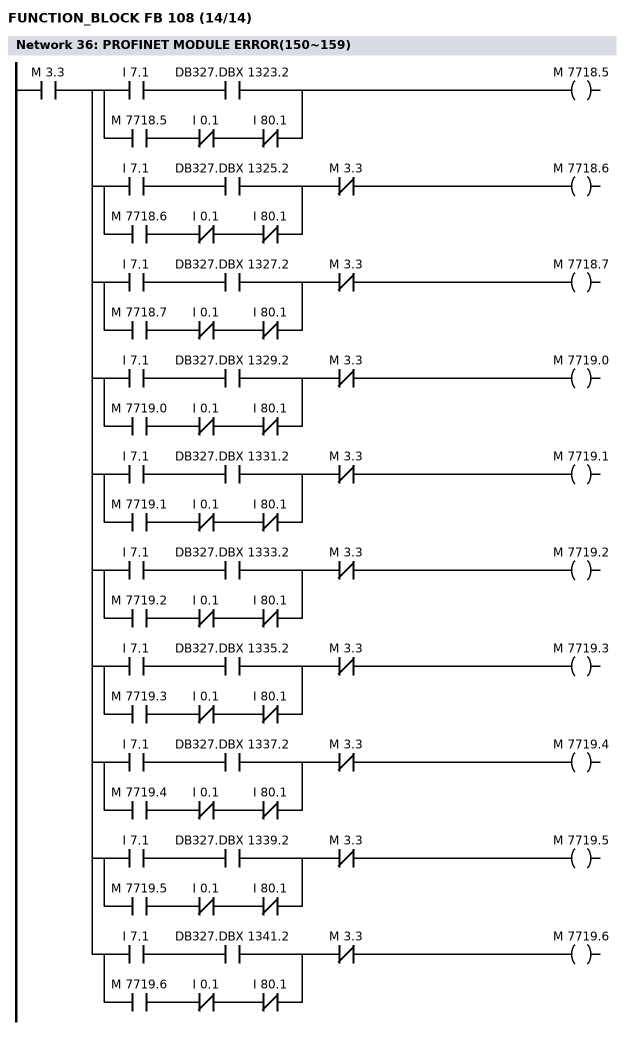

      A     M      3.3;
      =     L      0.0;
      A     L      0.0;
      A(    ;
      A     I      7.1;
      A     DB327.DBX 1323.2;
      O     ;
      A     M   7718.5;
      AN    I      0.1;
      AN    I     80.1;
      )     ;
      =     M   7718.5;
      A     L      0.0;
      A(    ;
      A     I      7.1;
      A     DB327.DBX 1325.2;
      O     ;
      A     M   7718.6;
      AN    I      0.1;
      AN    I     80.1;
      )     ;
      AN    M      3.3;
      =     M   7718.6;
      A     L      0.0;
      A(    ;
      A     I      7.1;
      A     DB327.DBX 1327.2;
      O     ;
      A     M   7718.7;
      AN    I      0.1;
      AN    I     80.1;
      )     ;
      AN    M      3.3;
      =     M   7718.7;
      A     L      0.0;
      A(    ;
      A     I      7.1;
      A     DB327.DBX 1329.2;
      O     ;
      A     M   7719.0;
      AN    I      0.1;
      AN    I     80.1;
      )     ;
      AN    M      3.3;
      =     M   7719.0;
      A     L      0.0;
      A(    ;
      A     I      7.1;
      A     DB327.DBX 1331.2;
      O     ;
      A     M   7719.1;
      AN    I      0.1;
      AN    I     80.1;
      )     ;
      AN    M      3.3;
      =     M   7719.1;
      A     L      0.0;
      A(    ;
      A     I      7.1;
      A     DB327.DBX 1333.2;
      O     ;
      A     M   7719.2;
      AN    I      0.1;
      AN    I     80.1;
      )     ;
      AN    M      3.3;
      =     M   7719.2;
      A     L      0.0;
      A(    ;
      A     I      7.1;
      A     DB327.DBX 1335.2;
      O     ;
      A     M   7719.3;
      AN    I      0.1;
      AN    I     80.1;
      )     ;
      AN    M      3.3;
      =     M   7719.3;
      A     L      0.0;
      A(    ;
      A     I      7.1;
      A     DB327.DBX 1337.2;
      O     ;
      A     M   7719.4;
      AN    I      0.1;
      AN    I     80.1;
      )     ;
      AN    M      3.3;
      =     M   7719.4;
      A     L      0.0;
      A(    ;
      A     I      7.1;
      A     DB327.DBX 1339.2;
      O     ;
      A     M   7719.5;
      AN    I      0.1;
      AN    I     80.1;
      )     ;
      AN    M      3.3;
      =     M   7719.5;
      A     L      0.0;
      A(    ;
      A     I      7.1;
      A     DB327.DBX 1341.2;
      O     ;
      A     M   7719.6;
      AN    I      0.1;
      AN    I     80.1;
      )     ;
      AN    M      3.3;
      =     M   7719.6;
END_FUNCTION_BLOCK

DATA_BLOCK DB 108
TITLE =
VERSION : 0.0

 FB 108
BEGIN
END_DATA_BLOCK

FUNCTION_BLOCK FB 110
TITLE =
VERSION : 0.1


VAR
  S705_MODE : FB 402;
END_VAR
BEGIN
NETWORK
TITLE =
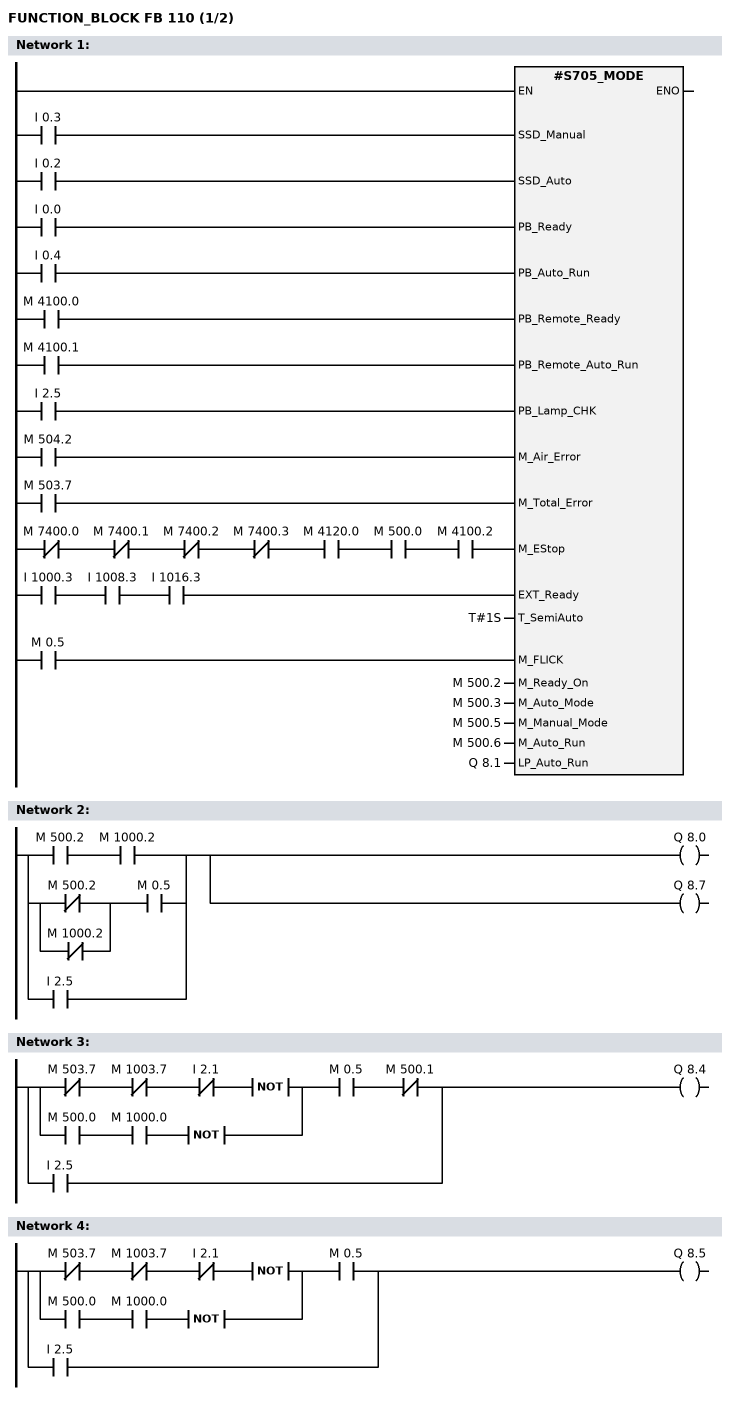

      A     I      0.3;
      =     L      0.0;
      BLD   103;
      A     I      0.2;
      =     L      0.1;
      BLD   103;
      A     I      0.0;
      =     L      0.2;
      BLD   103;
      A     I      0.4;
      =     L      0.3;
      BLD   103;
      A     M   4100.0;
      =     L      0.4;
      BLD   103;
      A     M   4100.1;
      =     L      0.5;
      BLD   103;
      A     I      2.5;
      =     L      0.6;
      BLD   103;
      A     M    504.2;
      =     L      0.7;
      BLD   103;
      A     M    503.7;
      =     L      1.1;
      BLD   103;
      AN    M   7400.0;
      AN    M   7400.1;
      AN    M   7400.2;
      AN    M   7400.3;
      A     M   4120.0;
      A     M    500.0;
      A     M   4100.2;
      =     L      1.2;
      BLD   103;
      A     I   1000.3;
      A     I   1008.3;
      A     I   1016.3;
      =     L      1.3;
      BLD   103;
      A     M      0.5;
      =     L      1.5;
      BLD   103;
      CALL #S705_MODE (
           SSD_Manual               := L      0.0,
           SSD_Auto                 := L      0.1,
           PB_Ready                 := L      0.2,
           PB_Auto_Run              := L      0.3,
           PB_Remote_Ready          := L      0.4,
           PB_Remote_Auto_Run       := L      0.5,
           PB_Lamp_CHK              := L      0.6,
           M_Air_Error              := L      0.7,
           M_Total_Error            := L      1.1,
           M_EStop                  := L      1.2,
           EXT_Ready                := L      1.3,
           T_SemiAuto               := T#1S,
           M_FLICK                  := L      1.5,
           M_Ready_On               := M    500.2,
           M_Auto_Mode              := M    500.3,
           M_Manual_Mode            := M    500.5,
           M_Auto_Run               := M    500.6,
           LP_Auto_Run              := Q      8.1);
      NOP   0;
NETWORK
TITLE =

      A     M    500.2;
      A     M   1000.2;
      O     ;
      A(    ;
      ON    M    500.2;
      ON    M   1000.2;
      )     ;
      A     M      0.5;
      O     I      2.5;
      =     Q      8.0;
      =     Q      8.7;
NETWORK
TITLE =

      A(    ;
      AN    M    503.7;
      AN    M   1003.7;
      AN    I      2.1;
      NOT   ;
      O(    ;
      A     M    500.0;
      A     M   1000.0;
      NOT   ;
      )     ;
      )     ;
      A     M      0.5;
      AN    M    500.1;
      O     I      2.5;
      =     Q      8.4;
NETWORK
TITLE =

      A(    ;
      AN    M    503.7;
      AN    M   1003.7;
      AN    I      2.1;
      NOT   ;
      O(    ;
      A     M    500.0;
      A     M   1000.0;
      NOT   ;
      )     ;
      )     ;
      A     M      0.5;
      O     I      2.5;
      =     Q      8.5;
NETWORK
TITLE =
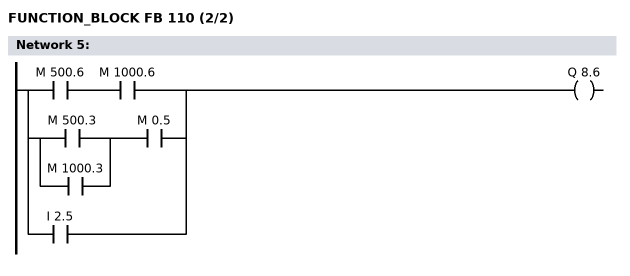

      A     M    500.6;
      A     M   1000.6;
      O     ;
      A(    ;
      O     M    500.3;
      O     M   1000.3;
      )     ;
      A     M      0.5;
      O     I      2.5;
      =     Q      8.6;
END_FUNCTION_BLOCK

DATA_BLOCK DB 110
TITLE =
VERSION : 0.0

 FB 110
BEGIN
   S705_MODE.SSD_Manual := FALSE;
   S705_MODE.SSD_Auto := TRUE;
   S705_MODE.PB_Ready := FALSE;
   S705_MODE.PB_Auto_Run := FALSE;
   S705_MODE.PB_Remote_Ready := FALSE;
   S705_MODE.PB_Remote_Auto_Run := FALSE;
   S705_MODE.PB_Lamp_CHK := FALSE;
   S705_MODE.M_Air_Error := FALSE;
   S705_MODE.M_Water_Error := FALSE;
   S705_MODE.M_Total_Error := FALSE;
   S705_MODE.M_EStop := TRUE;
   S705_MODE.EXT_Ready := TRUE;
   S705_MODE.EXT_Auto := FALSE;
   S705_MODE.T_SemiAuto := T#1S;
   S705_MODE.M_FLICK := TRUE;
   S705_MODE.M_Ready_On := TRUE;
   S705_MODE.M_Auto_Mode := TRUE;
   S705_MODE.M_SemiAuto_Mode := FALSE;
   S705_MODE.M_Manual_Mode := FALSE;
   S705_MODE.M_Auto_Run := TRUE;
   S705_MODE.LP_Ready_On := TRUE;
   S705_MODE.LP_Auto_Run := TRUE;
   S705_MODE.AUTO_MODE_DELAY.IN := FALSE;
   S705_MODE.AUTO_MODE_DELAY.PT := T#0MS;
   S705_MODE.AUTO_MODE_DELAY.Q := FALSE;
   S705_MODE.AUTO_MODE_DELAY.ET := T#0MS;
   S705_MODE.AUTO_MODE_DELAY.STATE := B#16#0;
   S705_MODE.AUTO_MODE_DELAY.STIME := T#0MS;
   S705_MODE.AUTO_MODE_DELAY.ATIME := T#0MS;
   S705_MODE.SEMI_AUTO_DELAY.IN := FALSE;
   S705_MODE.SEMI_AUTO_DELAY.PT := T#1S;
   S705_MODE.SEMI_AUTO_DELAY.Q := FALSE;
   S705_MODE.SEMI_AUTO_DELAY.ET := T#0MS;
   S705_MODE.SEMI_AUTO_DELAY.STATE := B#16#0;
   S705_MODE.SEMI_AUTO_DELAY.STIME := T#10D17H34M32S300MS;
   S705_MODE.SEMI_AUTO_DELAY.ATIME := T#10D17H34M32S323MS;
   S705_MODE.MANUAL_DELAY.IN := FALSE;
   S705_MODE.MANUAL_DELAY.PT := T#0MS;
   S705_MODE.MANUAL_DELAY.Q := FALSE;
   S705_MODE.MANUAL_DELAY.ET := T#0MS;
   S705_MODE.MANUAL_DELAY.STATE := B#16#0;
   S705_MODE.MANUAL_DELAY.STIME := T#0MS;
   S705_MODE.MANUAL_DELAY.ATIME := T#0MS;
END_DATA_BLOCK

FUNCTION FC 110 : VOID
TITLE =
VERSION : 0.1

BEGIN
NETWORK
TITLE =
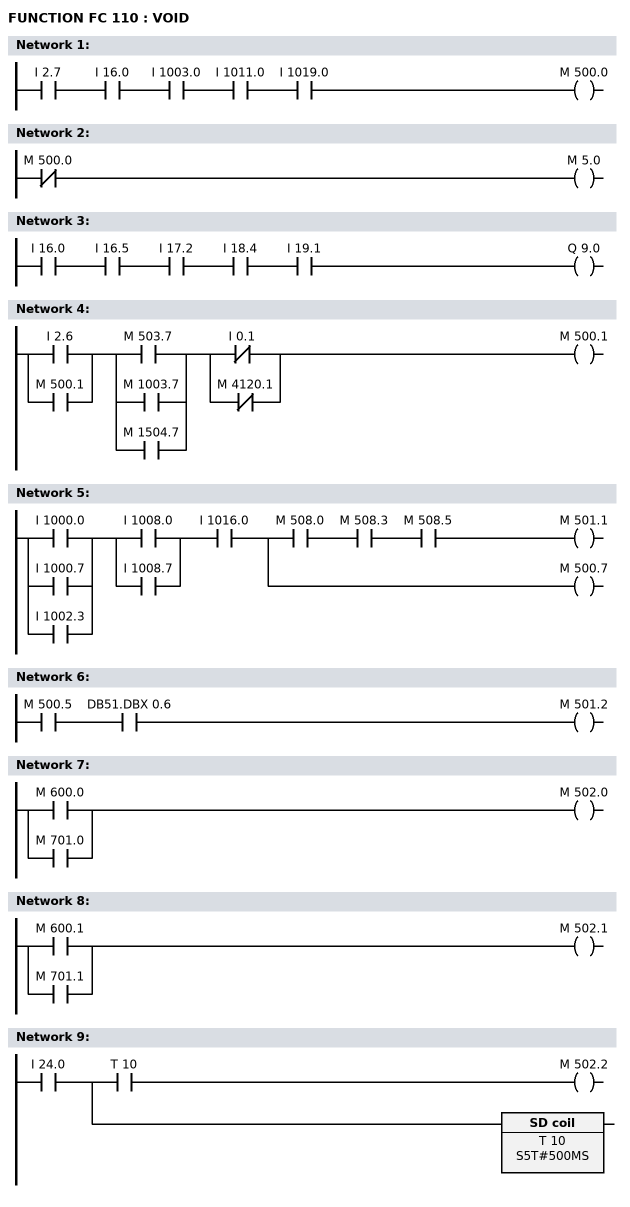

      A     I      2.7;
      A     I     16.0;
      A     I   1003.0;
      A     I   1011.0;
      A     I   1019.0;
      =     M    500.0;
NETWORK
TITLE =

      AN    M    500.0;
      =     M      5.0;
NETWORK
TITLE =

      A     I     16.0;
      A     I     16.5;
      A     I     17.2;
      A     I     18.4;
      A     I     19.1;
      =     Q      9.0;
NETWORK
TITLE =

      A(    ;
      O     I      2.6;
      O     M    500.1;
      )     ;
      A(    ;
      O     M    503.7;
      O     M   1003.7;
      O     M   1504.7;
      )     ;
      A(    ;
      ON    I      0.1;
      ON    M   4120.1;
      )     ;
      =     M    500.1;
NETWORK
TITLE =

      A(    ;
      O     I   1000.0;
      O     I   1000.7;
      O     I   1002.3;
      )     ;
      A(    ;
      O     I   1008.0;
      O     I   1008.7;
      )     ;
      A     I   1016.0;
      =     L      0.0;
      A     L      0.0;
      A     M    508.0;
      A     M    508.3;
      A     M    508.5;
      =     M    501.1;
      A     L      0.0;
      BLD   102;
      =     M    500.7;
NETWORK
TITLE =

      A     M    500.5;
      A     DB51.DBX    0.6;
      =     M    501.2;
NETWORK
TITLE =

      O     M    600.0;
      O     M    701.0;
      =     M    502.0;
NETWORK
TITLE =

      O     M    600.1;
      O     M    701.1;
      =     M    502.1;
NETWORK
TITLE =

      A     I     24.0;
      =     L      0.0;
      A     L      0.0;
      A     T     10;
      =     M    502.2;
      A     L      0.0;
      BLD   102;
      L     S5T#500MS;
      SD    T     10;
NETWORK
TITLE =

      AN    OV;
      A(    ;
      A     M    144.0;
      A     M    304.0;
      O     ;
      A     M    144.1;
      A     M    304.1;
      )     ;
      A(    ;
      A(    ;
      L     MD   140;
      L     MD   300;
      ==R   ;
      )     ;
      A(    ;
      L     MD   144;
      L     MD   304;
      ==R   ;
      )     ;
      A(    ;
      L     MD   148;
      L     MD   308;
      ==R   ;
      )     ;
      O     I      1.3;
      )     ;
      =     M    502.3;
NETWORK
TITLE =
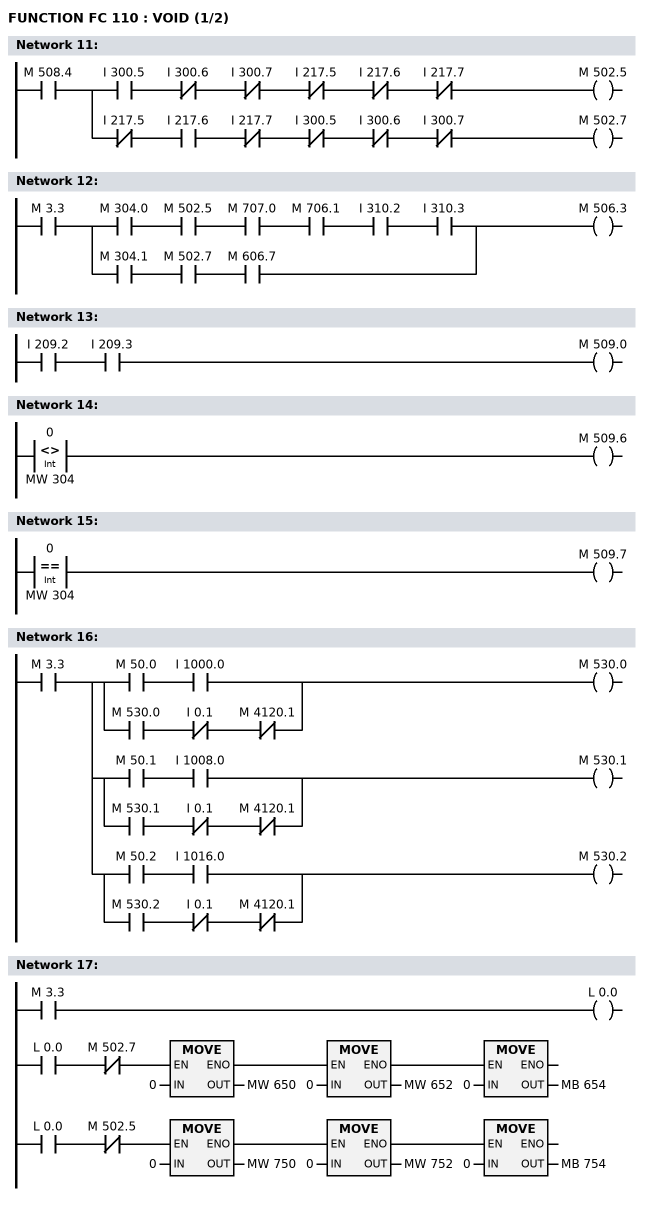

      A     M    508.4;
      =     L      0.0;
      A     L      0.0;
      A     I    300.5;
      AN    I    300.6;
      AN    I    300.7;
      AN    I    217.5;
      AN    I    217.6;
      AN    I    217.7;
      =     M    502.5;
      A     L      0.0;
      AN    I    217.5;
      A     I    217.6;
      AN    I    217.7;
      AN    I    300.5;
      AN    I    300.6;
      AN    I    300.7;
      =     M    502.7;
NETWORK
TITLE =

      A     M      3.3;
      A(    ;
      A     M    304.0;
      A     M    502.5;
      A     M    707.0;
      A     M    706.1;
      A     I    310.2;
      A     I    310.3;
      O     ;
      A     M    304.1;
      A     M    502.7;
      A     M    606.7;
      )     ;
      =     M    506.3;
NETWORK
TITLE =

      A     I    209.2;
      A     I    209.3;
      =     M    509.0;
NETWORK
TITLE =

      L     0;
      L     MW   304;
      <>I   ;
      =     M    509.6;
NETWORK
TITLE =

      L     0;
      L     MW   304;
      ==I   ;
      =     M    509.7;
NETWORK
TITLE =

      A     M      3.3;
      =     L      0.0;
      A     L      0.0;
      A(    ;
      A     M     50.0;
      A     I   1000.0;
      O     ;
      A     M    530.0;
      AN    I      0.1;
      AN    M   4120.1;
      )     ;
      =     M    530.0;
      A     L      0.0;
      A(    ;
      A     M     50.1;
      A     I   1008.0;
      O     ;
      A     M    530.1;
      AN    I      0.1;
      AN    M   4120.1;
      )     ;
      =     M    530.1;
      A     L      0.0;
      A(    ;
      A     M     50.2;
      A     I   1016.0;
      O     ;
      A     M    530.2;
      AN    I      0.1;
      AN    M   4120.1;
      )     ;
      =     M    530.2;
NETWORK
TITLE =

      A     M      3.3;
      =     L      0.0;
      A(    ;
      A(    ;
      A     L      0.0;
      AN    M    502.7;
      JNB   _001;
      L     0;
      T     MW   650;
      SET   ;
      SAVE  ;
      CLR   ;
_001: A     BR;
      )     ;
      JNB   _002;
      L     0;
      T     MW   652;
      SET   ;
      SAVE  ;
      CLR   ;
_002: A     BR;
      )     ;
      JNB   _003;
      L     0;
      T     MB   654;
_003: NOP   0;
      A(    ;
      A(    ;
      A     L      0.0;
      AN    M    502.5;
      JNB   _004;
      L     0;
      T     MW   750;
      SET   ;
      SAVE  ;
      CLR   ;
_004: A     BR;
      )     ;
      JNB   _005;
      L     0;
      T     MW   752;
      SET   ;
      SAVE  ;
      CLR   ;
_005: A     BR;
      )     ;
      JNB   _006;
      L     0;
      T     MB   754;
_006: NOP   0;
NETWORK
TITLE =
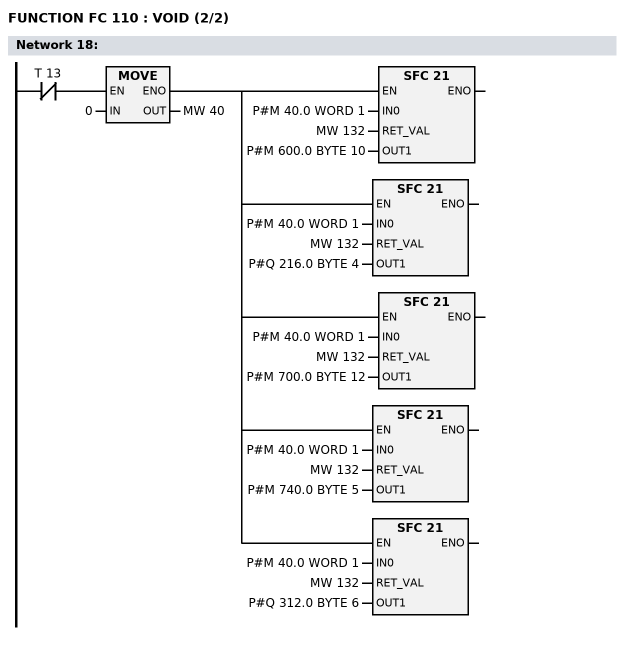

      AN    T     13;
      JNB   _007;
      L     0;
      T     MW    40;
      SET   ;
      SAVE  ;
      CLR   ;
_007: A     BR;
      =     L      0.0;
      A     L      0.0;
      JNB   _008;
      CALL SFC   21 (
           IN0                      := P#M 40.0 WORD 1,
           RET_VAL                  := MW   132,
           OUT1                     := P#M 600.0 BYTE 10);
_008: NOP   0;
      A     L      0.0;
      JNB   _009;
      CALL SFC   21 (
           IN0                      := P#M 40.0 WORD 1,
           RET_VAL                  := MW   132,
           OUT1                     := P#Q 216.0 BYTE 4);
_009: NOP   0;
      A     L      0.0;
      JNB   _00a;
      CALL SFC   21 (
           IN0                      := P#M 40.0 WORD 1,
           RET_VAL                  := MW   132,
           OUT1                     := P#M 700.0 BYTE 12);
_00a: NOP   0;
      A     L      0.0;
      JNB   _00b;
      CALL SFC   21 (
           IN0                      := P#M 40.0 WORD 1,
           RET_VAL                  := MW   132,
           OUT1                     := P#M 740.0 BYTE 5);
_00b: NOP   0;
      A     L      0.0;
      JNB   _00c;
      CALL SFC   21 (
           IN0                      := P#M 40.0 WORD 1,
           RET_VAL                  := MW   132,
           OUT1                     := P#Q 312.0 BYTE 6);
_00c: NOP   0;
END_FUNCTION

FUNCTION_BLOCK FB 111
TITLE =
VERSION : 0.1


VAR
  S705_HOOK_PIN : FB 424;
  S705_DC_LOCK : FB 424;
  S705_ELE : FB 424;
  S705_AIR_ELE : FB 424;
END_VAR
BEGIN
NETWORK
TITLE =
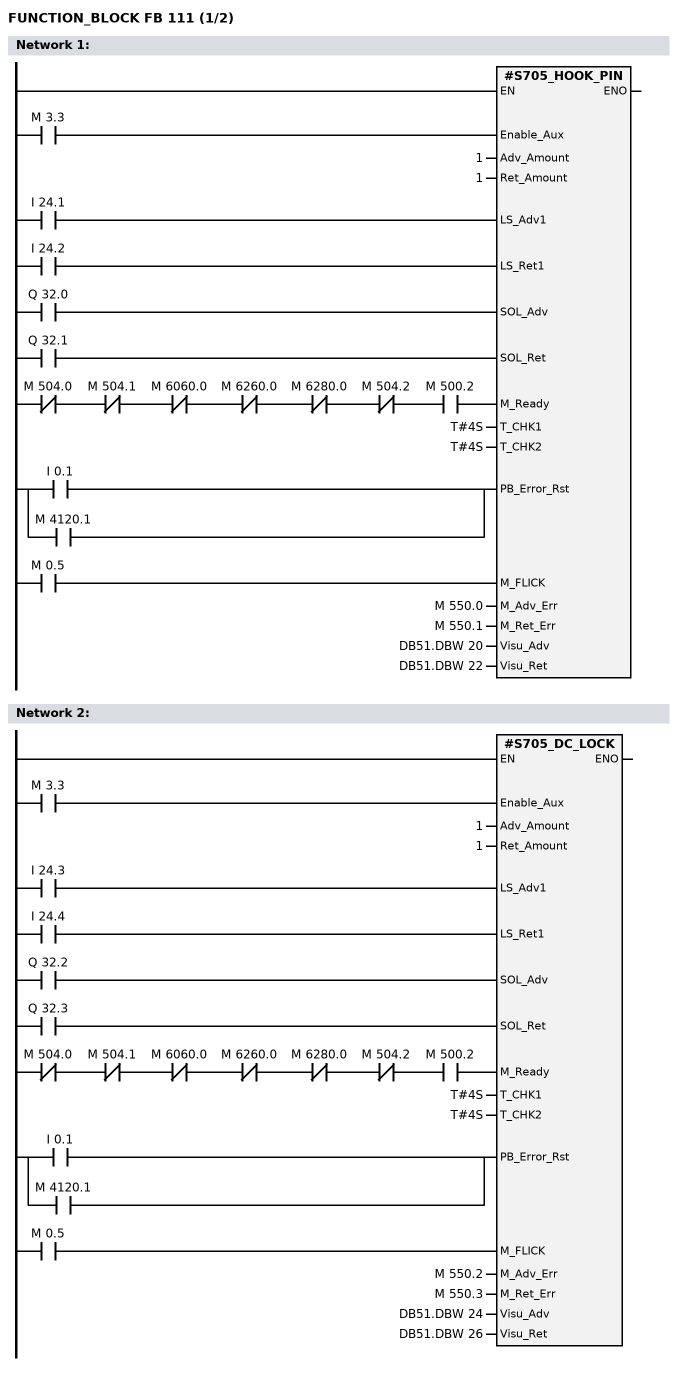

      A     M      3.3;
      =     L      0.0;
      BLD   103;
      A     I     24.1;
      =     L      0.1;
      BLD   103;
      A     I     24.2;
      =     L      0.2;
      BLD   103;
      A     Q     32.0;
      =     L      1.1;
      BLD   103;
      A     Q     32.1;
      =     L      1.2;
      BLD   103;
      AN    M    504.0;
      AN    M    504.1;
      AN    M   6060.0;
      AN    M   6260.0;
      AN    M   6280.0;
      AN    M    504.2;
      A     M    500.2;
      =     L      1.3;
      BLD   103;
      A(    ;
      O     I      0.1;
      O     M   4120.1;
      )     ;
      =     L      1.5;
      BLD   103;
      A     M      0.5;
      =     L      1.6;
      BLD   103;
      CALL #S705_HOOK_PIN (
           Enable_Aux               := L      0.0,
           Adv_Amount               := 1,
           Ret_Amount               := 1,
           LS_Adv1                  := L      0.1,
           LS_Ret1                  := L      0.2,
           SOL_Adv                  := L      1.1,
           SOL_Ret                  := L      1.2,
           M_Ready                  := L      1.3,
           T_CHK1                   := T#4S,
           T_CHK2                   := T#4S,
           PB_Error_Rst             := L      1.5,
           M_FLICK                  := L      1.6,
           M_Adv_Err                := M    550.0,
           M_Ret_Err                := M    550.1,
           Visu_Adv                 := DB51.DBW   20,
           Visu_Ret                 := DB51.DBW   22);
      NOP   0;
NETWORK
TITLE =

      A     M      3.3;
      =     L      0.0;
      BLD   103;
      A     I     24.3;
      =     L      0.1;
      BLD   103;
      A     I     24.4;
      =     L      0.2;
      BLD   103;
      A     Q     32.2;
      =     L      1.1;
      BLD   103;
      A     Q     32.3;
      =     L      1.2;
      BLD   103;
      AN    M    504.0;
      AN    M    504.1;
      AN    M   6060.0;
      AN    M   6260.0;
      AN    M   6280.0;
      AN    M    504.2;
      A     M    500.2;
      =     L      1.3;
      BLD   103;
      A(    ;
      O     I      0.1;
      O     M   4120.1;
      )     ;
      =     L      1.5;
      BLD   103;
      A     M      0.5;
      =     L      1.6;
      BLD   103;
      CALL #S705_DC_LOCK (
           Enable_Aux               := L      0.0,
           Adv_Amount               := 1,
           Ret_Amount               := 1,
           LS_Adv1                  := L      0.1,
           LS_Ret1                  := L      0.2,
           SOL_Adv                  := L      1.1,
           SOL_Ret                  := L      1.2,
           M_Ready                  := L      1.3,
           T_CHK1                   := T#4S,
           T_CHK2                   := T#4S,
           PB_Error_Rst             := L      1.5,
           M_FLICK                  := L      1.6,
           M_Adv_Err                := M    550.2,
           M_Ret_Err                := M    550.3,
           Visu_Adv                 := DB51.DBW   24,
           Visu_Ret                 := DB51.DBW   26);
      NOP   0;
NETWORK
TITLE =
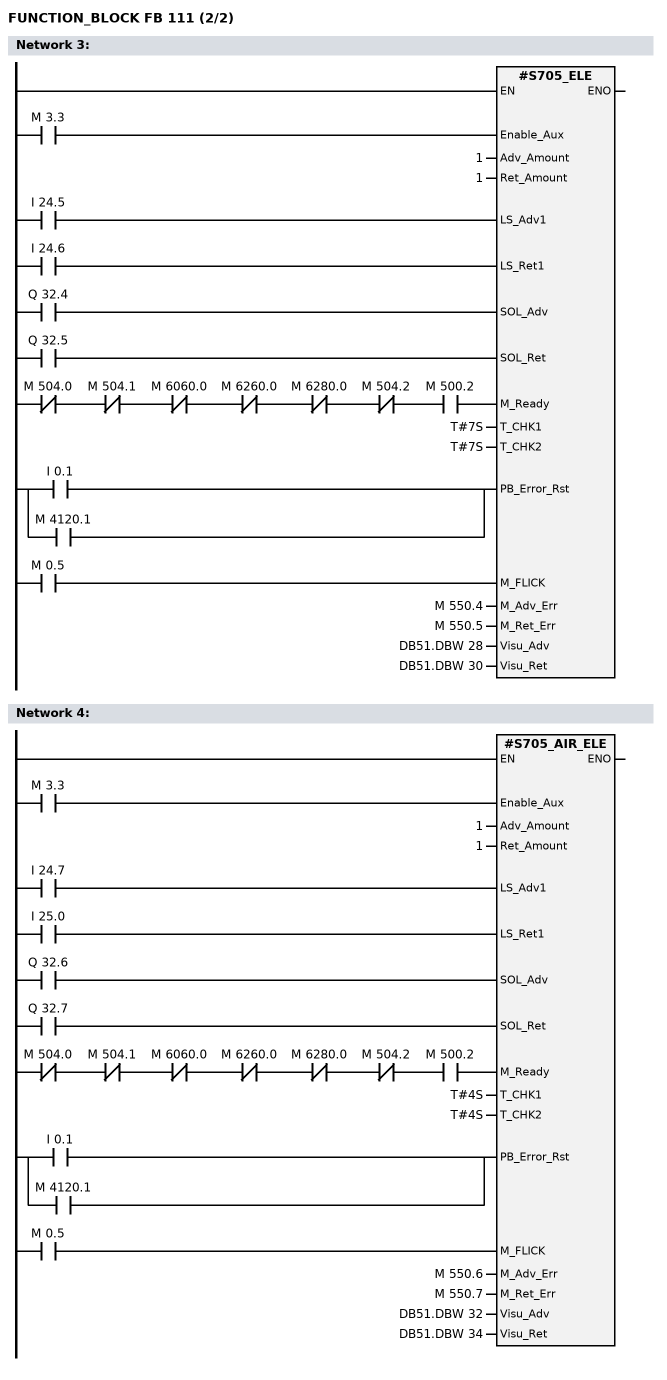

      A     M      3.3;
      =     L      0.0;
      BLD   103;
      A     I     24.5;
      =     L      0.1;
      BLD   103;
      A     I     24.6;
      =     L      0.2;
      BLD   103;
      A     Q     32.4;
      =     L      1.1;
      BLD   103;
      A     Q     32.5;
      =     L      1.2;
      BLD   103;
      AN    M    504.0;
      AN    M    504.1;
      AN    M   6060.0;
      AN    M   6260.0;
      AN    M   6280.0;
      AN    M    504.2;
      A     M    500.2;
      =     L      1.3;
      BLD   103;
      A(    ;
      O     I      0.1;
      O     M   4120.1;
      )     ;
      =     L      1.5;
      BLD   103;
      A     M      0.5;
      =     L      1.6;
      BLD   103;
      CALL #S705_ELE (
           Enable_Aux               := L      0.0,
           Adv_Amount               := 1,
           Ret_Amount               := 1,
           LS_Adv1                  := L      0.1,
           LS_Ret1                  := L      0.2,
           SOL_Adv                  := L      1.1,
           SOL_Ret                  := L      1.2,
           M_Ready                  := L      1.3,
           T_CHK1                   := T#7S,
           T_CHK2                   := T#7S,
           PB_Error_Rst             := L      1.5,
           M_FLICK                  := L      1.6,
           M_Adv_Err                := M    550.4,
           M_Ret_Err                := M    550.5,
           Visu_Adv                 := DB51.DBW   28,
           Visu_Ret                 := DB51.DBW   30);
      NOP   0;
NETWORK
TITLE =

      A     M      3.3;
      =     L      0.0;
      BLD   103;
      A     I     24.7;
      =     L      0.1;
      BLD   103;
      A     I     25.0;
      =     L      0.2;
      BLD   103;
      A     Q     32.6;
      =     L      1.1;
      BLD   103;
      A     Q     32.7;
      =     L      1.2;
      BLD   103;
      AN    M    504.0;
      AN    M    504.1;
      AN    M   6060.0;
      AN    M   6260.0;
      AN    M   6280.0;
      AN    M    504.2;
      A     M    500.2;
      =     L      1.3;
      BLD   103;
      A(    ;
      O     I      0.1;
      O     M   4120.1;
      )     ;
      =     L      1.5;
      BLD   103;
      A     M      0.5;
      =     L      1.6;
      BLD   103;
      CALL #S705_AIR_ELE (
           Enable_Aux               := L      0.0,
           Adv_Amount               := 1,
           Ret_Amount               := 1,
           LS_Adv1                  := L      0.1,
           LS_Ret1                  := L      0.2,
           SOL_Adv                  := L      1.1,
           SOL_Ret                  := L      1.2,
           M_Ready                  := L      1.3,
           T_CHK1                   := T#4S,
           T_CHK2                   := T#4S,
           PB_Error_Rst             := L      1.5,
           M_FLICK                  := L      1.6,
           M_Adv_Err                := M    550.6,
           M_Ret_Err                := M    550.7,
           Visu_Adv                 := DB51.DBW   32,
           Visu_Ret                 := DB51.DBW   34);
      NOP   0;
END_FUNCTION_BLOCK

DATA_BLOCK DB 111
TITLE =
VERSION : 0.0

 FB 111
BEGIN
   S705_HOOK_PIN.Enable_Aux := TRUE;
   S705_HOOK_PIN.Adv_Amount := 1;
   S705_HOOK_PIN.Ret_Amount := 1;
   S705_HOOK_PIN.LS_Adv1 := FALSE;
   S705_HOOK_PIN.LS_Ret1 := TRUE;
   S705_HOOK_PIN.LS_Adv2 := FALSE;
   S705_HOOK_PIN.LS_Ret2 := FALSE;
   S705_HOOK_PIN.LS_Adv3 := FALSE;
   S705_HOOK_PIN.LS_Ret3 := FALSE;
   S705_HOOK_PIN.LS_Adv4 := FALSE;
   S705_HOOK_PIN.LS_Ret4 := FALSE;
   S705_HOOK_PIN.SOL_Adv := FALSE;
   S705_HOOK_PIN.SOL_Ret := FALSE;
   S705_HOOK_PIN.M_Ready := TRUE;
   S705_HOOK_PIN.T_CHK1 := T#4S;
   S705_HOOK_PIN.T_CHK2 := T#4S;
   S705_HOOK_PIN.PB_Lamp_CHK := FALSE;
   S705_HOOK_PIN.PB_Error_Rst := FALSE;
   S705_HOOK_PIN.M_FLICK := FALSE;
   S705_HOOK_PIN.M_Adv_Err := FALSE;
   S705_HOOK_PIN.M_Ret_Err := FALSE;
   S705_HOOK_PIN.LP_Adv := FALSE;
   S705_HOOK_PIN.LP_Ret := TRUE;
   S705_HOOK_PIN.Visu_Adv := W#16#0;
   S705_HOOK_PIN.Visu_Ret := W#16#300;
   S705_HOOK_PIN.Error_T1.IN := FALSE;
   S705_HOOK_PIN.Error_T1.PT := T#4S;
   S705_HOOK_PIN.Error_T1.Q := FALSE;
   S705_HOOK_PIN.Error_T1.ET := T#0MS;
   S705_HOOK_PIN.Error_T1.STATE := B#16#0;
   S705_HOOK_PIN.Error_T1.STIME := T#23D5H8M43S362MS;
   S705_HOOK_PIN.Error_T1.ATIME := T#23D5H8M43S775MS;
   S705_HOOK_PIN.Error_T2.IN := FALSE;
   S705_HOOK_PIN.Error_T2.PT := T#4S;
   S705_HOOK_PIN.Error_T2.Q := FALSE;
   S705_HOOK_PIN.Error_T2.ET := T#0MS;
   S705_HOOK_PIN.Error_T2.STATE := B#16#0;
   S705_HOOK_PIN.Error_T2.STIME := T#0MS;
   S705_HOOK_PIN.Error_T2.ATIME := T#0MS;
   S705_HOOK_PIN.CHK_Aux1 := FALSE;
   S705_HOOK_PIN.CHK_Aux2 := FALSE;
   S705_HOOK_PIN.Error_T1_DN := FALSE;
   S705_HOOK_PIN.Error_T2_DN := FALSE;
   S705_HOOK_PIN.Adv_Memo := FALSE;
   S705_HOOK_PIN.Visu_Adv_Arr[0] := FALSE;
   S705_HOOK_PIN.Visu_Adv_Arr[1] := FALSE;
   S705_HOOK_PIN.Visu_Adv_Arr[2] := FALSE;
   S705_HOOK_PIN.Visu_Adv_Arr[3] := FALSE;
   S705_HOOK_PIN.Visu_Adv_Arr[4] := FALSE;
   S705_HOOK_PIN.Visu_Adv_Arr[5] := FALSE;
   S705_HOOK_PIN.Visu_Adv_Arr[6] := FALSE;
   S705_HOOK_PIN.Visu_Adv_Arr[7] := FALSE;
   S705_HOOK_PIN.Visu_Adv_Arr[8] := FALSE;
   S705_HOOK_PIN.Visu_Adv_Arr[9] := FALSE;
   S705_HOOK_PIN.Visu_Adv_Arr[10] := FALSE;
   S705_HOOK_PIN.Visu_Adv_Arr[11] := FALSE;
   S705_HOOK_PIN.Visu_Adv_Arr[12] := FALSE;
   S705_HOOK_PIN.Visu_Adv_Arr[13] := FALSE;
   S705_HOOK_PIN.Visu_Adv_Arr[14] := FALSE;
   S705_HOOK_PIN.Visu_Adv_Arr[15] := FALSE;
   S705_HOOK_PIN.Visu_Ret_Arr[0] := TRUE;
   S705_HOOK_PIN.Visu_Ret_Arr[1] := TRUE;
   S705_HOOK_PIN.Visu_Ret_Arr[2] := FALSE;
   S705_HOOK_PIN.Visu_Ret_Arr[3] := FALSE;
   S705_HOOK_PIN.Visu_Ret_Arr[4] := FALSE;
   S705_HOOK_PIN.Visu_Ret_Arr[5] := FALSE;
   S705_HOOK_PIN.Visu_Ret_Arr[6] := FALSE;
   S705_HOOK_PIN.Visu_Ret_Arr[7] := FALSE;
   S705_HOOK_PIN.Visu_Ret_Arr[8] := FALSE;
   S705_HOOK_PIN.Visu_Ret_Arr[9] := FALSE;
   S705_HOOK_PIN.Visu_Ret_Arr[10] := FALSE;
   S705_HOOK_PIN.Visu_Ret_Arr[11] := FALSE;
   S705_HOOK_PIN.Visu_Ret_Arr[12] := FALSE;
   S705_HOOK_PIN.Visu_Ret_Arr[13] := FALSE;
   S705_HOOK_PIN.Visu_Ret_Arr[14] := FALSE;
   S705_HOOK_PIN.Visu_Ret_Arr[15] := FALSE;
   S705_HOOK_PIN.BLK_Move_Ret := 0;
   S705_HOOK_PIN.Enable := TRUE;
   S705_HOOK_PIN.Adv_End := FALSE;
   S705_HOOK_PIN.Ret_End := TRUE;
   S705_DC_LOCK.Enable_Aux := TRUE;
   S705_DC_LOCK.Adv_Amount := 1;
   S705_DC_LOCK.Ret_Amount := 1;
   S705_DC_LOCK.LS_Adv1 := TRUE;
   S705_DC_LOCK.LS_Ret1 := FALSE;
   S705_DC_LOCK.LS_Adv2 := FALSE;
   S705_DC_LOCK.LS_Ret2 := FALSE;
   S705_DC_LOCK.LS_Adv3 := FALSE;
   S705_DC_LOCK.LS_Ret3 := FALSE;
   S705_DC_LOCK.LS_Adv4 := FALSE;
   S705_DC_LOCK.LS_Ret4 := FALSE;
   S705_DC_LOCK.SOL_Adv := FALSE;
   S705_DC_LOCK.SOL_Ret := FALSE;
   S705_DC_LOCK.M_Ready := TRUE;
   S705_DC_LOCK.T_CHK1 := T#4S;
   S705_DC_LOCK.T_CHK2 := T#4S;
   S705_DC_LOCK.PB_Lamp_CHK := FALSE;
   S705_DC_LOCK.PB_Error_Rst := FALSE;
   S705_DC_LOCK.M_FLICK := FALSE;
   S705_DC_LOCK.M_Adv_Err := FALSE;
   S705_DC_LOCK.M_Ret_Err := FALSE;
   S705_DC_LOCK.LP_Adv := TRUE;
   S705_DC_LOCK.LP_Ret := FALSE;
   S705_DC_LOCK.Visu_Adv := W#16#300;
   S705_DC_LOCK.Visu_Ret := W#16#0;
   S705_DC_LOCK.Error_T1.IN := FALSE;
   S705_DC_LOCK.Error_T1.PT := T#4S;
   S705_DC_LOCK.Error_T1.Q := FALSE;
   S705_DC_LOCK.Error_T1.ET := T#0MS;
   S705_DC_LOCK.Error_T1.STATE := B#16#0;
   S705_DC_LOCK.Error_T1.STIME := T#23D5H8M43S362MS;
   S705_DC_LOCK.Error_T1.ATIME := T#23D5H8M44S6MS;
   S705_DC_LOCK.Error_T2.IN := FALSE;
   S705_DC_LOCK.Error_T2.PT := T#4S;
   S705_DC_LOCK.Error_T2.Q := FALSE;
   S705_DC_LOCK.Error_T2.ET := T#0MS;
   S705_DC_LOCK.Error_T2.STATE := B#16#0;
   S705_DC_LOCK.Error_T2.STIME := T#0MS;
   S705_DC_LOCK.Error_T2.ATIME := T#0MS;
   S705_DC_LOCK.CHK_Aux1 := FALSE;
   S705_DC_LOCK.CHK_Aux2 := FALSE;
   S705_DC_LOCK.Error_T1_DN := FALSE;
   S705_DC_LOCK.Error_T2_DN := FALSE;
   S705_DC_LOCK.Adv_Memo := TRUE;
   S705_DC_LOCK.Visu_Adv_Arr[0] := TRUE;
   S705_DC_LOCK.Visu_Adv_Arr[1] := TRUE;
   S705_DC_LOCK.Visu_Adv_Arr[2] := FALSE;
   S705_DC_LOCK.Visu_Adv_Arr[3] := FALSE;
   S705_DC_LOCK.Visu_Adv_Arr[4] := FALSE;
   S705_DC_LOCK.Visu_Adv_Arr[5] := FALSE;
   S705_DC_LOCK.Visu_Adv_Arr[6] := FALSE;
   S705_DC_LOCK.Visu_Adv_Arr[7] := FALSE;
   S705_DC_LOCK.Visu_Adv_Arr[8] := FALSE;
   S705_DC_LOCK.Visu_Adv_Arr[9] := FALSE;
   S705_DC_LOCK.Visu_Adv_Arr[10] := FALSE;
   S705_DC_LOCK.Visu_Adv_Arr[11] := FALSE;
   S705_DC_LOCK.Visu_Adv_Arr[12] := FALSE;
   S705_DC_LOCK.Visu_Adv_Arr[13] := FALSE;
   S705_DC_LOCK.Visu_Adv_Arr[14] := FALSE;
   S705_DC_LOCK.Visu_Adv_Arr[15] := FALSE;
   S705_DC_LOCK.Visu_Ret_Arr[0] := FALSE;
   S705_DC_LOCK.Visu_Ret_Arr[1] := FALSE;
   S705_DC_LOCK.Visu_Ret_Arr[2] := FALSE;
   S705_DC_LOCK.Visu_Ret_Arr[3] := FALSE;
   S705_DC_LOCK.Visu_Ret_Arr[4] := FALSE;
   S705_DC_LOCK.Visu_Ret_Arr[5] := FALSE;
   S705_DC_LOCK.Visu_Ret_Arr[6] := FALSE;
   S705_DC_LOCK.Visu_Ret_Arr[7] := FALSE;
   S705_DC_LOCK.Visu_Ret_Arr[8] := FALSE;
   S705_DC_LOCK.Visu_Ret_Arr[9] := FALSE;
   S705_DC_LOCK.Visu_Ret_Arr[10] := FALSE;
   S705_DC_LOCK.Visu_Ret_Arr[11] := FALSE;
   S705_DC_LOCK.Visu_Ret_Arr[12] := FALSE;
   S705_DC_LOCK.Visu_Ret_Arr[13] := FALSE;
   S705_DC_LOCK.Visu_Ret_Arr[14] := FALSE;
   S705_DC_LOCK.Visu_Ret_Arr[15] := FALSE;
   S705_DC_LOCK.BLK_Move_Ret := 0;
   S705_DC_LOCK.Enable := TRUE;
   S705_DC_LOCK.Adv_End := TRUE;
   S705_DC_LOCK.Ret_End := FALSE;
   S705_ELE.Enable_Aux := TRUE;
   S705_ELE.Adv_Amount := 1;
   S705_ELE.Ret_Amount := 1;
   S705_ELE.LS_Adv1 := TRUE;
   S705_ELE.LS_Ret1 := FALSE;
   S705_ELE.LS_Adv2 := FALSE;
   S705_ELE.LS_Ret2 := FALSE;
   S705_ELE.LS_Adv3 := FALSE;
   S705_ELE.LS_Ret3 := FALSE;
   S705_ELE.LS_Adv4 := FALSE;
   S705_ELE.LS_Ret4 := FALSE;
   S705_ELE.SOL_Adv := FALSE;
   S705_ELE.SOL_Ret := FALSE;
   S705_ELE.M_Ready := TRUE;
   S705_ELE.T_CHK1 := T#7S;
   S705_ELE.T_CHK2 := T#7S;
   S705_ELE.PB_Lamp_CHK := FALSE;
   S705_ELE.PB_Error_Rst := FALSE;
   S705_ELE.M_FLICK := FALSE;
   S705_ELE.M_Adv_Err := FALSE;
   S705_ELE.M_Ret_Err := FALSE;
   S705_ELE.LP_Adv := TRUE;
   S705_ELE.LP_Ret := FALSE;
   S705_ELE.Visu_Adv := W#16#300;
   S705_ELE.Visu_Ret := W#16#0;
   S705_ELE.Error_T1.IN := FALSE;
   S705_ELE.Error_T1.PT := T#7S;
   S705_ELE.Error_T1.Q := FALSE;
   S705_ELE.Error_T1.ET := T#0MS;
   S705_ELE.Error_T1.STATE := B#16#0;
   S705_ELE.Error_T1.STIME := T#23D5H8M44S538MS;
   S705_ELE.Error_T1.ATIME := T#23D5H8M44S923MS;
   S705_ELE.Error_T2.IN := FALSE;
   S705_ELE.Error_T2.PT := T#7S;
   S705_ELE.Error_T2.Q := FALSE;
   S705_ELE.Error_T2.ET := T#0MS;
   S705_ELE.Error_T2.STATE := B#16#0;
   S705_ELE.Error_T2.STIME := T#0MS;
   S705_ELE.Error_T2.ATIME := T#0MS;
   S705_ELE.CHK_Aux1 := FALSE;
   S705_ELE.CHK_Aux2 := FALSE;
   S705_ELE.Error_T1_DN := FALSE;
   S705_ELE.Error_T2_DN := FALSE;
   S705_ELE.Adv_Memo := TRUE;
   S705_ELE.Visu_Adv_Arr[0] := TRUE;
   S705_ELE.Visu_Adv_Arr[1] := TRUE;
   S705_ELE.Visu_Adv_Arr[2] := FALSE;
   S705_ELE.Visu_Adv_Arr[3] := FALSE;
   S705_ELE.Visu_Adv_Arr[4] := FALSE;
   S705_ELE.Visu_Adv_Arr[5] := FALSE;
   S705_ELE.Visu_Adv_Arr[6] := FALSE;
   S705_ELE.Visu_Adv_Arr[7] := FALSE;
   S705_ELE.Visu_Adv_Arr[8] := FALSE;
   S705_ELE.Visu_Adv_Arr[9] := FALSE;
   S705_ELE.Visu_Adv_Arr[10] := FALSE;
   S705_ELE.Visu_Adv_Arr[11] := FALSE;
   S705_ELE.Visu_Adv_Arr[12] := FALSE;
   S705_ELE.Visu_Adv_Arr[13] := FALSE;
   S705_ELE.Visu_Adv_Arr[14] := FALSE;
   S705_ELE.Visu_Adv_Arr[15] := FALSE;
   S705_ELE.Visu_Ret_Arr[0] := FALSE;
   S705_ELE.Visu_Ret_Arr[1] := FALSE;
   S705_ELE.Visu_Ret_Arr[2] := FALSE;
   S705_ELE.Visu_Ret_Arr[3] := FALSE;
   S705_ELE.Visu_Ret_Arr[4] := FALSE;
   S705_ELE.Visu_Ret_Arr[5] := FALSE;
   S705_ELE.Visu_Ret_Arr[6] := FALSE;
   S705_ELE.Visu_Ret_Arr[7] := FALSE;
   S705_ELE.Visu_Ret_Arr[8] := FALSE;
   S705_ELE.Visu_Ret_Arr[9] := FALSE;
   S705_ELE.Visu_Ret_Arr[10] := FALSE;
   S705_ELE.Visu_Ret_Arr[11] := FALSE;
   S705_ELE.Visu_Ret_Arr[12] := FALSE;
   S705_ELE.Visu_Ret_Arr[13] := FALSE;
   S705_ELE.Visu_Ret_Arr[14] := FALSE;
   S705_ELE.Visu_Ret_Arr[15] := FALSE;
   S705_ELE.BLK_Move_Ret := 0;
   S705_ELE.Enable := TRUE;
   S705_ELE.Adv_End := TRUE;
   S705_ELE.Ret_End := FALSE;
   S705_AIR_ELE.Enable_Aux := TRUE;
   S705_AIR_ELE.Adv_Amount := 1;
   S705_AIR_ELE.Ret_Amount := 1;
   S705_AIR_ELE.LS_Adv1 := TRUE;
   S705_AIR_ELE.LS_Ret1 := FALSE;
   S705_AIR_ELE.LS_Adv2 := FALSE;
   S705_AIR_ELE.LS_Ret2 := FALSE;
   S705_AIR_ELE.LS_Adv3 := FALSE;
   S705_AIR_ELE.LS_Ret3 := FALSE;
   S705_AIR_ELE.LS_Adv4 := FALSE;
   S705_AIR_ELE.LS_Ret4 := FALSE;
   S705_AIR_ELE.SOL_Adv := FALSE;
   S705_AIR_ELE.SOL_Ret := FALSE;
   S705_AIR_ELE.M_Ready := TRUE;
   S705_AIR_ELE.T_CHK1 := T#4S;
   S705_AIR_ELE.T_CHK2 := T#4S;
   S705_AIR_ELE.PB_Lamp_CHK := FALSE;
   S705_AIR_ELE.PB_Error_Rst := FALSE;
   S705_AIR_ELE.M_FLICK := FALSE;
   S705_AIR_ELE.M_Adv_Err := FALSE;
   S705_AIR_ELE.M_Ret_Err := FALSE;
   S705_AIR_ELE.LP_Adv := TRUE;
   S705_AIR_ELE.LP_Ret := FALSE;
   S705_AIR_ELE.Visu_Adv := W#16#300;
   S705_AIR_ELE.Visu_Ret := W#16#0;
   S705_AIR_ELE.Error_T1.IN := FALSE;
   S705_AIR_ELE.Error_T1.PT := T#4S;
   S705_AIR_ELE.Error_T1.Q := FALSE;
   S705_AIR_ELE.Error_T1.ET := T#0MS;
   S705_AIR_ELE.Error_T1.STATE := B#16#0;
   S705_AIR_ELE.Error_T1.STIME := T#23D5H8M44S538MS;
   S705_AIR_ELE.Error_T1.ATIME := T#23D5H8M44S606MS;
   S705_AIR_ELE.Error_T2.IN := FALSE;
   S705_AIR_ELE.Error_T2.PT := T#4S;
   S705_AIR_ELE.Error_T2.Q := FALSE;
   S705_AIR_ELE.Error_T2.ET := T#0MS;
   S705_AIR_ELE.Error_T2.STATE := B#16#0;
   S705_AIR_ELE.Error_T2.STIME := T#0MS;
   S705_AIR_ELE.Error_T2.ATIME := T#0MS;
   S705_AIR_ELE.CHK_Aux1 := FALSE;
   S705_AIR_ELE.CHK_Aux2 := FALSE;
   S705_AIR_ELE.Error_T1_DN := FALSE;
   S705_AIR_ELE.Error_T2_DN := FALSE;
   S705_AIR_ELE.Adv_Memo := TRUE;
   S705_AIR_ELE.Visu_Adv_Arr[0] := TRUE;
   S705_AIR_ELE.Visu_Adv_Arr[1] := TRUE;
   S705_AIR_ELE.Visu_Adv_Arr[2] := FALSE;
   S705_AIR_ELE.Visu_Adv_Arr[3] := FALSE;
   S705_AIR_ELE.Visu_Adv_Arr[4] := FALSE;
   S705_AIR_ELE.Visu_Adv_Arr[5] := FALSE;
   S705_AIR_ELE.Visu_Adv_Arr[6] := FALSE;
   S705_AIR_ELE.Visu_Adv_Arr[7] := FALSE;
   S705_AIR_ELE.Visu_Adv_Arr[8] := FALSE;
   S705_AIR_ELE.Visu_Adv_Arr[9] := FALSE;
   S705_AIR_ELE.Visu_Adv_Arr[10] := FALSE;
   S705_AIR_ELE.Visu_Adv_Arr[11] := FALSE;
   S705_AIR_ELE.Visu_Adv_Arr[12] := FALSE;
   S705_AIR_ELE.Visu_Adv_Arr[13] := FALSE;
   S705_AIR_ELE.Visu_Adv_Arr[14] := FALSE;
   S705_AIR_ELE.Visu_Adv_Arr[15] := FALSE;
   S705_AIR_ELE.Visu_Ret_Arr[0] := FALSE;
   S705_AIR_ELE.Visu_Ret_Arr[1] := FALSE;
   S705_AIR_ELE.Visu_Ret_Arr[2] := FALSE;
   S705_AIR_ELE.Visu_Ret_Arr[3] := FALSE;
   S705_AIR_ELE.Visu_Ret_Arr[4] := FALSE;
   S705_AIR_ELE.Visu_Ret_Arr[5] := FALSE;
   S705_AIR_ELE.Visu_Ret_Arr[6] := FALSE;
   S705_AIR_ELE.Visu_Ret_Arr[7] := FALSE;
   S705_AIR_ELE.Visu_Ret_Arr[8] := FALSE;
   S705_AIR_ELE.Visu_Ret_Arr[9] := FALSE;
   S705_AIR_ELE.Visu_Ret_Arr[10] := FALSE;
   S705_AIR_ELE.Visu_Ret_Arr[11] := FALSE;
   S705_AIR_ELE.Visu_Ret_Arr[12] := FALSE;
   S705_AIR_ELE.Visu_Ret_Arr[13] := FALSE;
   S705_AIR_ELE.Visu_Ret_Arr[14] := FALSE;
   S705_AIR_ELE.Visu_Ret_Arr[15] := FALSE;
   S705_AIR_ELE.BLK_Move_Ret := 0;
   S705_AIR_ELE.Enable := TRUE;
   S705_AIR_ELE.Adv_End := TRUE;
   S705_AIR_ELE.Ret_End := FALSE;
END_DATA_BLOCK

FUNCTION FC 111 : VOID
TITLE =
VERSION : 0.1

BEGIN
NETWORK
TITLE =
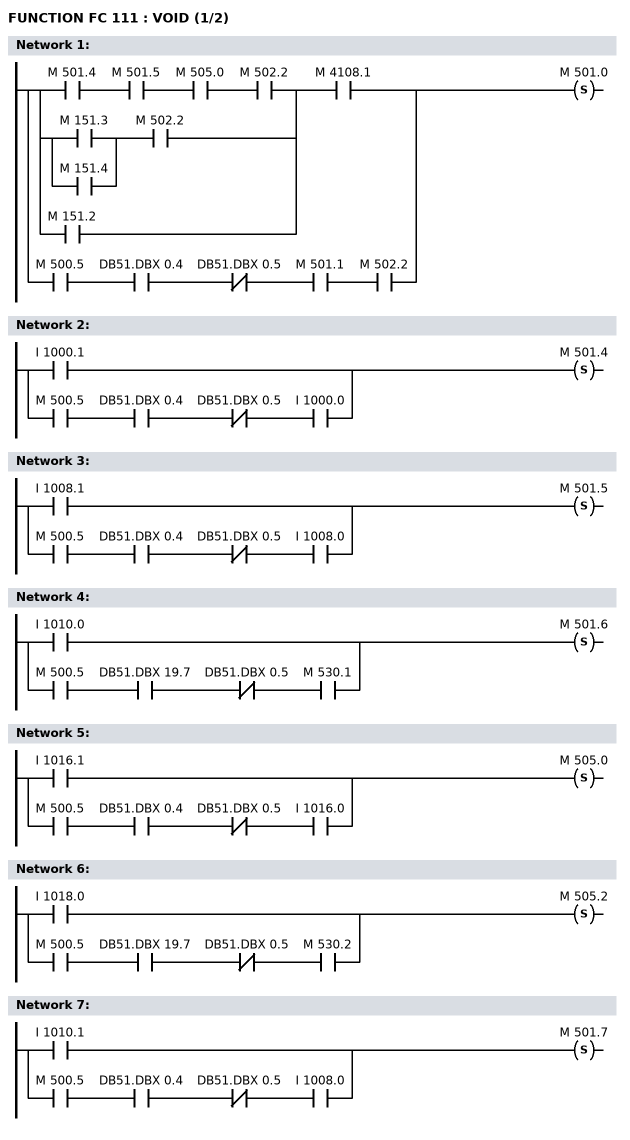

      A(    ;
      A     M    501.4;
      A     M    501.5;
      A     M    505.0;
      A     M    502.2;
      O     ;
      A(    ;
      O     M    151.3;
      O     M    151.4;
      )     ;
      A     M    502.2;
      O     M    151.2;
      )     ;
      A     M   4108.1;
      O     ;
      A     M    500.5;
      A     DB51.DBX    0.4;
      AN    DB51.DBX    0.5;
      A     M    501.1;
      A     M    502.2;
      S     M    501.0;
NETWORK
TITLE =

      O     I   1000.1;
      O     ;
      A     M    500.5;
      A     DB51.DBX    0.4;
      AN    DB51.DBX    0.5;
      A     I   1000.0;
      S     M    501.4;
NETWORK
TITLE =

      O     I   1008.1;
      O     ;
      A     M    500.5;
      A     DB51.DBX    0.4;
      AN    DB51.DBX    0.5;
      A     I   1008.0;
      S     M    501.5;
NETWORK
TITLE =

      O     I   1010.0;
      O     ;
      A     M    500.5;
      A     DB51.DBX   19.7;
      AN    DB51.DBX    0.5;
      A     M    530.1;
      S     M    501.6;
NETWORK
TITLE =

      O     I   1016.1;
      O     ;
      A     M    500.5;
      A     DB51.DBX    0.4;
      AN    DB51.DBX    0.5;
      A     I   1016.0;
      S     M    505.0;
NETWORK
TITLE =

      O     I   1018.0;
      O     ;
      A     M    500.5;
      A     DB51.DBX   19.7;
      AN    DB51.DBX    0.5;
      A     M    530.2;
      S     M    505.2;
NETWORK
TITLE =

      O     I   1010.1;
      O     ;
      A     M    500.5;
      A     DB51.DBX    0.4;
      AN    DB51.DBX    0.5;
      A     I   1008.0;
      S     M    501.7;
NETWORK
TITLE =
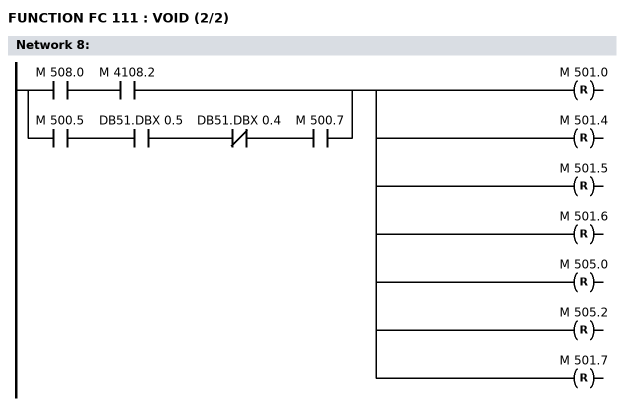

      A     M    508.0;
      A     M   4108.2;
      O     ;
      A     M    500.5;
      A     DB51.DBX    0.5;
      AN    DB51.DBX    0.4;
      A     M    500.7;
      R     M    501.0;
      R     M    501.4;
      R     M    501.5;
      R     M    501.6;
      R     M    505.0;
      R     M    505.2;
      R     M    501.7;
END_FUNCTION

FUNCTION_BLOCK FB 112
TITLE =
VERSION : 0.1

BEGIN
NETWORK
TITLE =
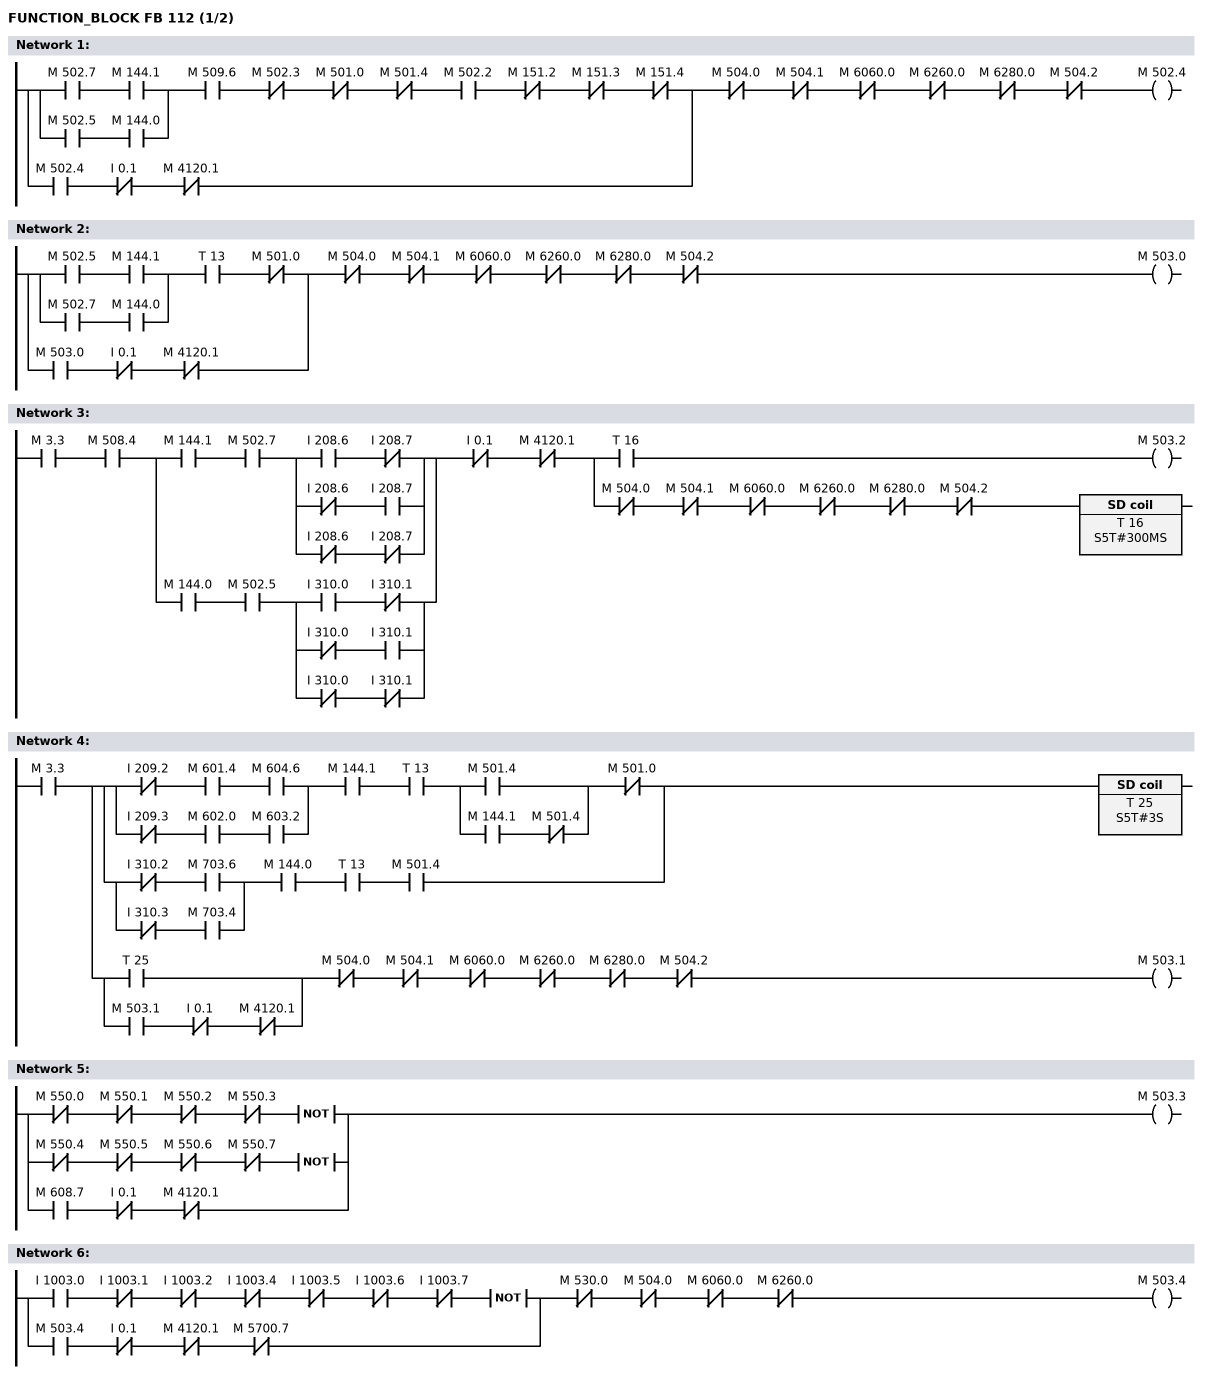

      A(    ;
      A(    ;
      A     M    502.7;
      A     M    144.1;
      O     ;
      A     M    502.5;
      A     M    144.0;
      )     ;
      A     M    509.6;
      AN    M    502.3;
      AN    M    501.0;
      AN    M    501.4;
      A     M    502.2;
      AN    M    151.2;
      AN    M    151.3;
      AN    M    151.4;
      O     ;
      A     M    502.4;
      AN    I      0.1;
      AN    M   4120.1;
      )     ;
      AN    M    504.0;
      AN    M    504.1;
      AN    M   6060.0;
      AN    M   6260.0;
      AN    M   6280.0;
      AN    M    504.2;
      =     M    502.4;
NETWORK
TITLE =

      A(    ;
      A(    ;
      A     M    502.5;
      A     M    144.1;
      O     ;
      A     M    502.7;
      A     M    144.0;
      )     ;
      A     T     13;
      AN    M    501.0;
      O     ;
      A     M    503.0;
      AN    I      0.1;
      AN    M   4120.1;
      )     ;
      AN    M    504.0;
      AN    M    504.1;
      AN    M   6060.0;
      AN    M   6260.0;
      AN    M   6280.0;
      AN    M    504.2;
      =     M    503.0;
NETWORK
TITLE =

      A     M      3.3;
      A     M    508.4;
      A(    ;
      A     M    144.1;
      A     M    502.7;
      A(    ;
      A     I    208.6;
      AN    I    208.7;
      O     ;
      AN    I    208.6;
      A     I    208.7;
      O     ;
      AN    I    208.6;
      AN    I    208.7;
      )     ;
      O     ;
      A     M    144.0;
      A     M    502.5;
      A(    ;
      A     I    310.0;
      AN    I    310.1;
      O     ;
      AN    I    310.0;
      A     I    310.1;
      O     ;
      AN    I    310.0;
      AN    I    310.1;
      )     ;
      )     ;
      AN    I      0.1;
      AN    M   4120.1;
      =     L      0.0;
      A     L      0.0;
      A     T     16;
      =     M    503.2;
      A     L      0.0;
      AN    M    504.0;
      AN    M    504.1;
      AN    M   6060.0;
      AN    M   6260.0;
      AN    M   6280.0;
      AN    M    504.2;
      L     S5T#300MS;
      SD    T     16;
NETWORK
TITLE =

      A     M      3.3;
      =     L      0.0;
      A     L      0.0;
      A(    ;
      A(    ;
      AN    I    209.2;
      A     M    601.4;
      A     M    604.6;
      O     ;
      AN    I    209.3;
      A     M    602.0;
      A     M    603.2;
      )     ;
      A     M    144.1;
      A     T     13;
      A(    ;
      O     M    501.4;
      O     ;
      A     M    144.1;
      AN    M    501.4;
      )     ;
      AN    M    501.0;
      O     ;
      A(    ;
      AN    I    310.2;
      A     M    703.6;
      O     ;
      AN    I    310.3;
      A     M    703.4;
      )     ;
      A     M    144.0;
      A     T     13;
      A     M    501.4;
      )     ;
      L     S5T#3S;
      SD    T     25;
      A     L      0.0;
      A(    ;
      O     T     25;
      O     ;
      A     M    503.1;
      AN    I      0.1;
      AN    M   4120.1;
      )     ;
      AN    M    504.0;
      AN    M    504.1;
      AN    M   6060.0;
      AN    M   6260.0;
      AN    M   6280.0;
      AN    M    504.2;
      =     M    503.1;
NETWORK
TITLE =

      AN    M    550.0;
      AN    M    550.1;
      AN    M    550.2;
      AN    M    550.3;
      NOT   ;
      O(    ;
      AN    M    550.4;
      AN    M    550.5;
      AN    M    550.6;
      AN    M    550.7;
      NOT   ;
      )     ;
      O     ;
      A     M    608.7;
      AN    I      0.1;
      AN    M   4120.1;
      =     M    503.3;
NETWORK
TITLE =

      A(    ;
      A     I   1003.0;
      AN    I   1003.1;
      AN    I   1003.2;
      AN    I   1003.4;
      AN    I   1003.5;
      AN    I   1003.6;
      AN    I   1003.7;
      NOT   ;
      O     ;
      A     M    503.4;
      AN    I      0.1;
      AN    M   4120.1;
      AN    M   5700.7;
      )     ;
      AN    M    530.0;
      AN    M    504.0;
      AN    M   6060.0;
      AN    M   6260.0;
      =     M    503.4;
NETWORK
TITLE =
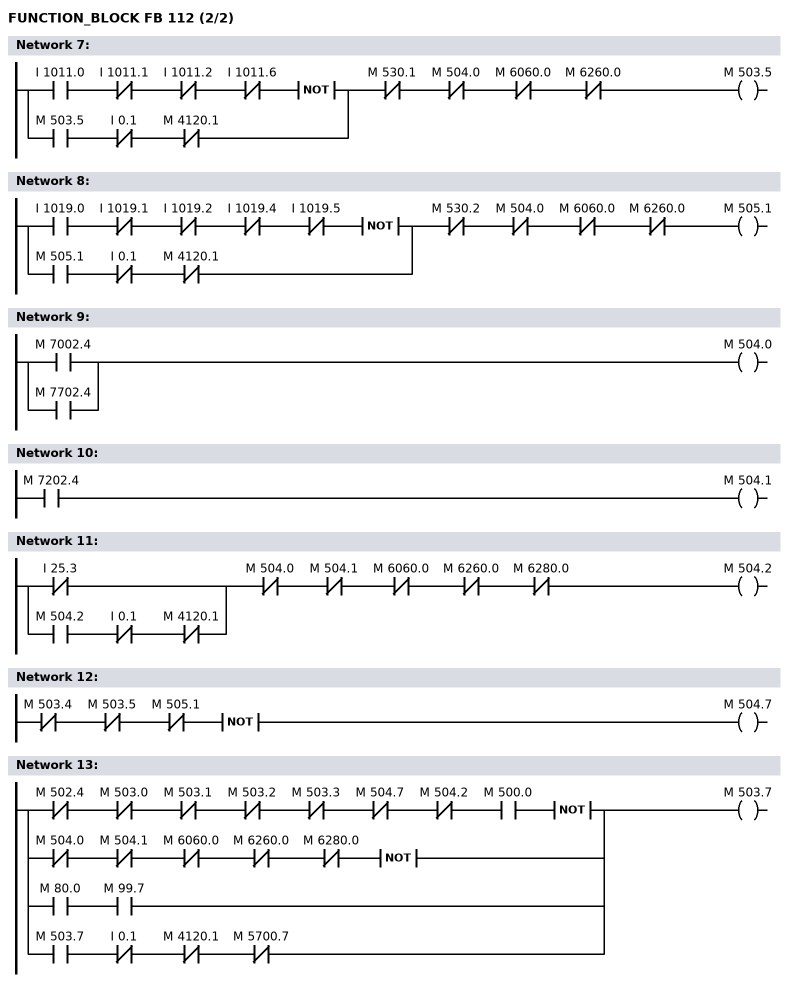

      A(    ;
      A     I   1011.0;
      AN    I   1011.1;
      AN    I   1011.2;
      AN    I   1011.6;
      NOT   ;
      O     ;
      A     M    503.5;
      AN    I      0.1;
      AN    M   4120.1;
      )     ;
      AN    M    530.1;
      AN    M    504.0;
      AN    M   6060.0;
      AN    M   6260.0;
      =     M    503.5;
NETWORK
TITLE =

      A(    ;
      A     I   1019.0;
      AN    I   1019.1;
      AN    I   1019.2;
      AN    I   1019.4;
      AN    I   1019.5;
      NOT   ;
      O     ;
      A     M    505.1;
      AN    I      0.1;
      AN    M   4120.1;
      )     ;
      AN    M    530.2;
      AN    M    504.0;
      AN    M   6060.0;
      AN    M   6260.0;
      =     M    505.1;
NETWORK
TITLE =

      O     M   7002.4;
      O     M   7702.4;
      =     M    504.0;
NETWORK
TITLE =

      A     M   7202.4;
      =     M    504.1;
NETWORK
TITLE =

      A(    ;
      ON    I     25.3;
      O     ;
      A     M    504.2;
      AN    I      0.1;
      AN    M   4120.1;
      )     ;
      AN    M    504.0;
      AN    M    504.1;
      AN    M   6060.0;
      AN    M   6260.0;
      AN    M   6280.0;
      =     M    504.2;
NETWORK
TITLE =

      AN    M    503.4;
      AN    M    503.5;
      AN    M    505.1;
      NOT   ;
      =     M    504.7;
NETWORK
TITLE =

      AN    M    502.4;
      AN    M    503.0;
      AN    M    503.1;
      AN    M    503.2;
      AN    M    503.3;
      AN    M    504.7;
      AN    M    504.2;
      A     M    500.0;
      NOT   ;
      O(    ;
      AN    M    504.0;
      AN    M    504.1;
      AN    M   6060.0;
      AN    M   6260.0;
      AN    M   6280.0;
      NOT   ;
      )     ;
      O     ;
      A     M     80.0;
      A     M     99.7;
      O     ;
      A     M    503.7;
      AN    I      0.1;
      AN    M   4120.1;
      AN    M   5700.7;
      =     M    503.7;
END_FUNCTION_BLOCK

DATA_BLOCK DB 112
TITLE =
VERSION : 0.0

 FB 112
BEGIN
END_DATA_BLOCK

FUNCTION FC 112 : VOID
TITLE =
VERSION : 0.1

BEGIN
NETWORK
TITLE =
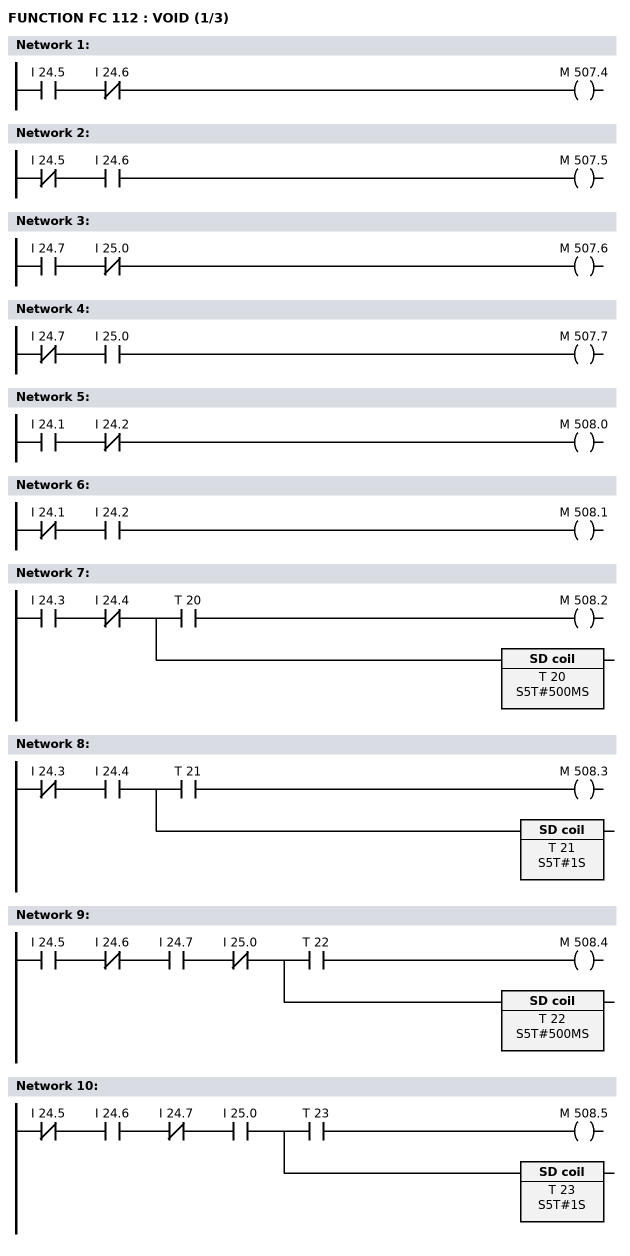

      A     I     24.5;
      AN    I     24.6;
      =     M    507.4;
NETWORK
TITLE =

      AN    I     24.5;
      A     I     24.6;
      =     M    507.5;
NETWORK
TITLE =

      A     I     24.7;
      AN    I     25.0;
      =     M    507.6;
NETWORK
TITLE =

      AN    I     24.7;
      A     I     25.0;
      =     M    507.7;
NETWORK
TITLE =

      A     I     24.1;
      AN    I     24.2;
      =     M    508.0;
NETWORK
TITLE =

      AN    I     24.1;
      A     I     24.2;
      =     M    508.1;
NETWORK
TITLE =

      A     I     24.3;
      AN    I     24.4;
      =     L      0.0;
      A     L      0.0;
      A     T     20;
      =     M    508.2;
      A     L      0.0;
      BLD   102;
      L     S5T#500MS;
      SD    T     20;
NETWORK
TITLE =

      AN    I     24.3;
      A     I     24.4;
      =     L      0.0;
      A     L      0.0;
      A     T     21;
      =     M    508.3;
      A     L      0.0;
      BLD   102;
      L     S5T#1S;
      SD    T     21;
NETWORK
TITLE =

      A     I     24.5;
      AN    I     24.6;
      A     I     24.7;
      AN    I     25.0;
      =     L      0.0;
      A     L      0.0;
      A     T     22;
      =     M    508.4;
      A     L      0.0;
      BLD   102;
      L     S5T#500MS;
      SD    T     22;
NETWORK
TITLE =

      AN    I     24.5;
      A     I     24.6;
      AN    I     24.7;
      A     I     25.0;
      =     L      0.0;
      A     L      0.0;
      A     T     23;
      =     M    508.5;
      A     L      0.0;
      BLD   102;
      L     S5T#1S;
      SD    T     23;
NETWORK
TITLE =#705 급전POWER전원
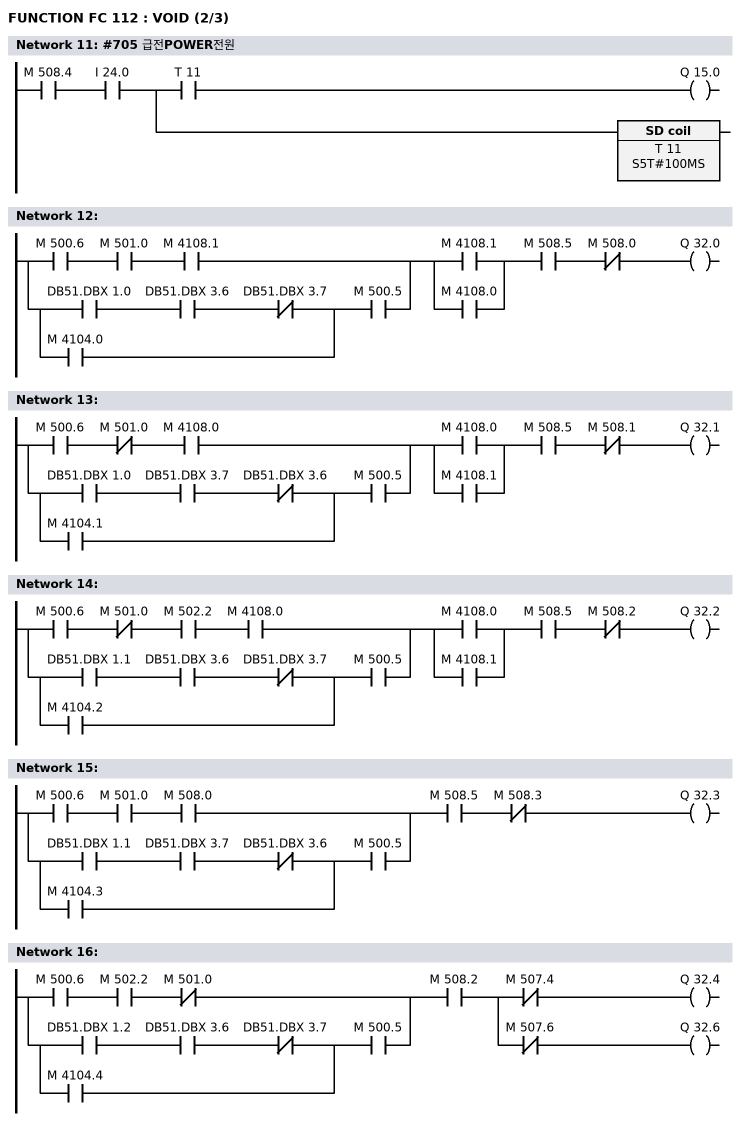

      A     M    508.4;
      A     I     24.0;
      =     L      0.0;
      A     L      0.0;
      A     T     11;
      =     Q     15.0;
      A     L      0.0;
      BLD   102;
      L     S5T#100MS;
      SD    T     11;
NETWORK
TITLE =

      A(    ;
      A     M    500.6;
      A     M    501.0;
      A     M   4108.1;
      O     ;
      A(    ;
      A     DB51.DBX    1.0;
      A     DB51.DBX    3.6;
      AN    DB51.DBX    3.7;
      O     M   4104.0;
      )     ;
      A     M    500.5;
      )     ;
      A(    ;
      O     M   4108.1;
      O     M   4108.0;
      )     ;
      A     M    508.5;
      AN    M    508.0;
      =     Q     32.0;
NETWORK
TITLE =

      A(    ;
      A     M    500.6;
      AN    M    501.0;
      A     M   4108.0;
      O     ;
      A(    ;
      A     DB51.DBX    1.0;
      A     DB51.DBX    3.7;
      AN    DB51.DBX    3.6;
      O     M   4104.1;
      )     ;
      A     M    500.5;
      )     ;
      A(    ;
      O     M   4108.0;
      O     M   4108.1;
      )     ;
      A     M    508.5;
      AN    M    508.1;
      =     Q     32.1;
NETWORK
TITLE =

      A(    ;
      A     M    500.6;
      AN    M    501.0;
      A     M    502.2;
      A     M   4108.0;
      O     ;
      A(    ;
      A     DB51.DBX    1.1;
      A     DB51.DBX    3.6;
      AN    DB51.DBX    3.7;
      O     M   4104.2;
      )     ;
      A     M    500.5;
      )     ;
      A(    ;
      O     M   4108.0;
      O     M   4108.1;
      )     ;
      A     M    508.5;
      AN    M    508.2;
      =     Q     32.2;
NETWORK
TITLE =

      A(    ;
      A     M    500.6;
      A     M    501.0;
      A     M    508.0;
      O     ;
      A(    ;
      A     DB51.DBX    1.1;
      A     DB51.DBX    3.7;
      AN    DB51.DBX    3.6;
      O     M   4104.3;
      )     ;
      A     M    500.5;
      )     ;
      A     M    508.5;
      AN    M    508.3;
      =     Q     32.3;
NETWORK
TITLE =

      A(    ;
      A     M    500.6;
      A     M    502.2;
      AN    M    501.0;
      O     ;
      A(    ;
      A     DB51.DBX    1.2;
      A     DB51.DBX    3.6;
      AN    DB51.DBX    3.7;
      O     M   4104.4;
      )     ;
      A     M    500.5;
      )     ;
      A     M    508.2;
      =     L      0.0;
      A     L      0.0;
      AN    M    507.4;
      =     Q     32.4;
      A     L      0.0;
      AN    M    507.6;
      =     Q     32.6;
NETWORK
TITLE =
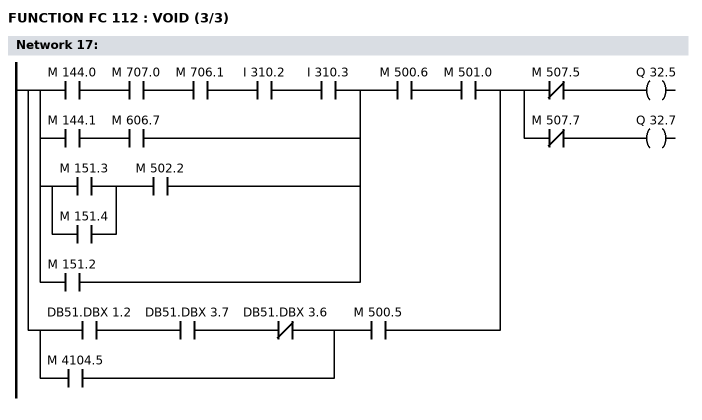

      A(    ;
      A     M    144.0;
      A     M    707.0;
      A     M    706.1;
      A     I    310.2;
      A     I    310.3;
      O     ;
      A     M    144.1;
      A     M    606.7;
      O     ;
      A(    ;
      O     M    151.3;
      O     M    151.4;
      )     ;
      A     M    502.2;
      O     M    151.2;
      )     ;
      A     M    500.6;
      A     M    501.0;
      O     ;
      A(    ;
      A     DB51.DBX    1.2;
      A     DB51.DBX    3.7;
      AN    DB51.DBX    3.6;
      O     M   4104.5;
      )     ;
      A     M    500.5;
      =     L      0.0;
      A     L      0.0;
      AN    M    507.5;
      =     Q     32.5;
      A     L      0.0;
      AN    M    507.7;
      =     Q     32.7;
END_FUNCTION

FUNCTION_BLOCK FB 113
TITLE =
VERSION : 0.1


VAR
  S705_LM_DC_PIN : FB 424;
  S705_LM_DC_1ST_CLAMP1 : FB 424;
  S705_LM_DC_1ST_CLAMP2 : FB 424;
  S705_LM_DC_1ST_CLAMP3 : FB 424;
  S705_LM_DC_1ST_CLAMP4 : FB 424;
  S705_LM_DC_2ND_CLAMP1 : FB 424;
  S705_LM_DC_2ND_CLAMP2 : FB 424;
  S705_LM_DC_2ND_CLAMP3 : FB 424;
  S705_LM_DC_2ND_CLAMP4 : FB 424;
  S705_LM_DC_2ND_CLAMP5 : FB 424;
  S705_LM_DC_STK_PIN : FB 424;
  S705_LM_DC_OTR_CLAMP : FB 424;
  S705_LM_DC_ASSY_CLAMP : FB 424;
  S705_LM_DC_FF_PIN : FB 424;
  S705_LM_DC_FF_CLAMP : FB 424;
  S705_LM_DC_2ND_CLAMP6 : FB 424;
  S705_LM_DC_2ND_CLAMP7 : FB 424;
  S705_LM_DC_1ST_CLAMP5 : FB 424;
END_VAR
BEGIN
NETWORK
TITLE =
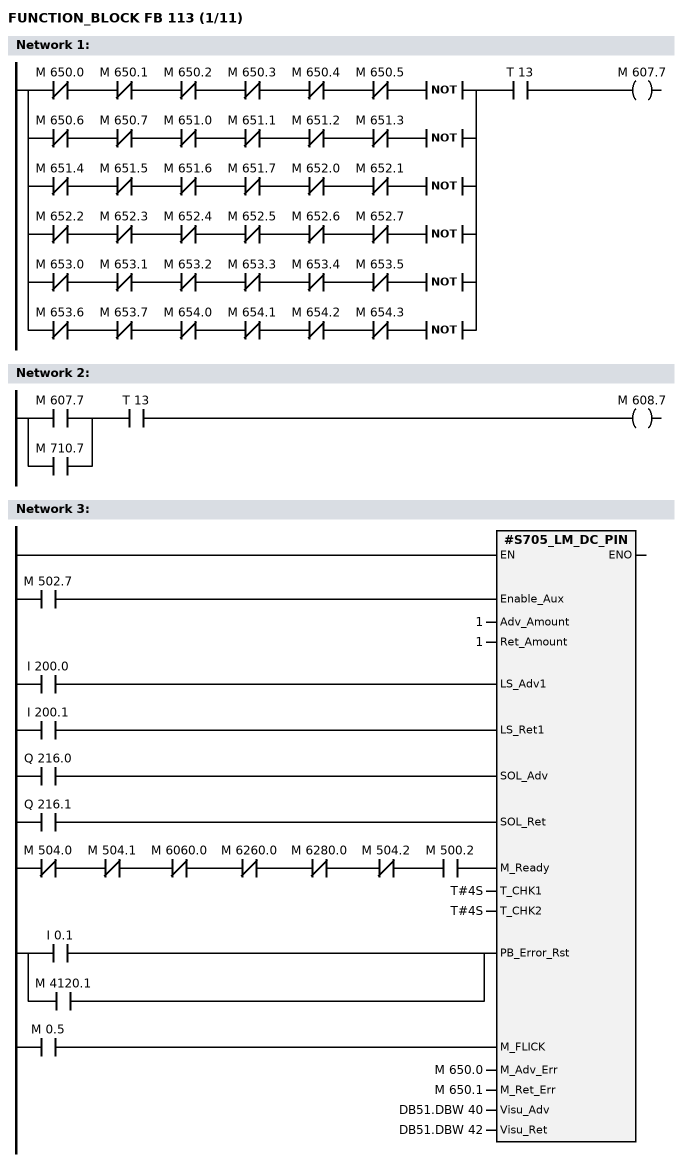

      A(    ;
      AN    M    650.0;
      AN    M    650.1;
      AN    M    650.2;
      AN    M    650.3;
      AN    M    650.4;
      AN    M    650.5;
      NOT   ;
      O(    ;
      AN    M    650.6;
      AN    M    650.7;
      AN    M    651.0;
      AN    M    651.1;
      AN    M    651.2;
      AN    M    651.3;
      NOT   ;
      )     ;
      O(    ;
      AN    M    651.4;
      AN    M    651.5;
      AN    M    651.6;
      AN    M    651.7;
      AN    M    652.0;
      AN    M    652.1;
      NOT   ;
      )     ;
      O(    ;
      AN    M    652.2;
      AN    M    652.3;
      AN    M    652.4;
      AN    M    652.5;
      AN    M    652.6;
      AN    M    652.7;
      NOT   ;
      )     ;
      O(    ;
      AN    M    653.0;
      AN    M    653.1;
      AN    M    653.2;
      AN    M    653.3;
      AN    M    653.4;
      AN    M    653.5;
      NOT   ;
      )     ;
      O(    ;
      AN    M    653.6;
      AN    M    653.7;
      AN    M    654.0;
      AN    M    654.1;
      AN    M    654.2;
      AN    M    654.3;
      NOT   ;
      )     ;
      )     ;
      A     T     13;
      =     M    607.7;
NETWORK
TITLE =

      A(    ;
      O     M    607.7;
      O     M    710.7;
      )     ;
      A     T     13;
      =     M    608.7;
NETWORK
TITLE =

      A     M    502.7;
      =     L      0.0;
      BLD   103;
      A     I    200.0;
      =     L      0.1;
      BLD   103;
      A     I    200.1;
      =     L      0.2;
      BLD   103;
      A     Q    216.0;
      =     L      1.1;
      BLD   103;
      A     Q    216.1;
      =     L      1.2;
      BLD   103;
      AN    M    504.0;
      AN    M    504.1;
      AN    M   6060.0;
      AN    M   6260.0;
      AN    M   6280.0;
      AN    M    504.2;
      A     M    500.2;
      =     L      1.3;
      BLD   103;
      A(    ;
      O     I      0.1;
      O     M   4120.1;
      )     ;
      =     L      1.5;
      BLD   103;
      A     M      0.5;
      =     L      1.6;
      BLD   103;
      CALL #S705_LM_DC_PIN (
           Enable_Aux               := L      0.0,
           Adv_Amount               := 1,
           Ret_Amount               := 1,
           LS_Adv1                  := L      0.1,
           LS_Ret1                  := L      0.2,
           SOL_Adv                  := L      1.1,
           SOL_Ret                  := L      1.2,
           M_Ready                  := L      1.3,
           T_CHK1                   := T#4S,
           T_CHK2                   := T#4S,
           PB_Error_Rst             := L      1.5,
           M_FLICK                  := L      1.6,
           M_Adv_Err                := M    650.0,
           M_Ret_Err                := M    650.1,
           Visu_Adv                 := DB51.DBW   40,
           Visu_Ret                 := DB51.DBW   42);
      NOP   0;
NETWORK
TITLE =
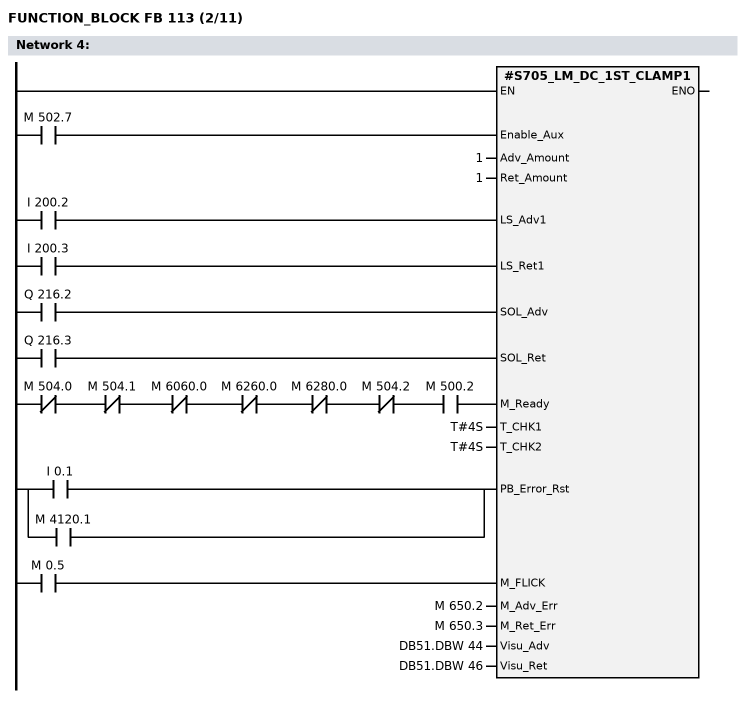

      A     M    502.7;
      =     L      0.0;
      BLD   103;
      A     I    200.2;
      =     L      0.1;
      BLD   103;
      A     I    200.3;
      =     L      0.2;
      BLD   103;
      A     Q    216.2;
      =     L      1.1;
      BLD   103;
      A     Q    216.3;
      =     L      1.2;
      BLD   103;
      AN    M    504.0;
      AN    M    504.1;
      AN    M   6060.0;
      AN    M   6260.0;
      AN    M   6280.0;
      AN    M    504.2;
      A     M    500.2;
      =     L      1.3;
      BLD   103;
      A(    ;
      O     I      0.1;
      O     M   4120.1;
      )     ;
      =     L      1.5;
      BLD   103;
      A     M      0.5;
      =     L      1.6;
      BLD   103;
      CALL #S705_LM_DC_1ST_CLAMP1 (
           Enable_Aux               := L      0.0,
           Adv_Amount               := 1,
           Ret_Amount               := 1,
           LS_Adv1                  := L      0.1,
           LS_Ret1                  := L      0.2,
           SOL_Adv                  := L      1.1,
           SOL_Ret                  := L      1.2,
           M_Ready                  := L      1.3,
           T_CHK1                   := T#4S,
           T_CHK2                   := T#4S,
           PB_Error_Rst             := L      1.5,
           M_FLICK                  := L      1.6,
           M_Adv_Err                := M    650.2,
           M_Ret_Err                := M    650.3,
           Visu_Adv                 := DB51.DBW   44,
           Visu_Ret                 := DB51.DBW   46);
      NOP   0;
NETWORK
TITLE =
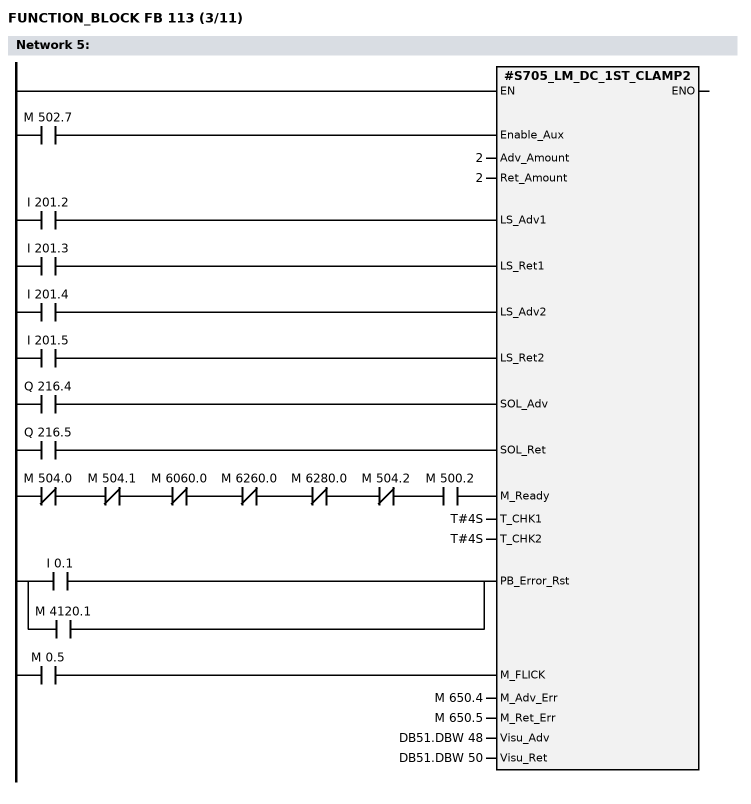

      A     M    502.7;
      =     L      0.0;
      BLD   103;
      A     I    201.2;
      =     L      0.1;
      BLD   103;
      A     I    201.3;
      =     L      0.2;
      BLD   103;
      A     I    201.4;
      =     L      0.3;
      BLD   103;
      A     I    201.5;
      =     L      0.4;
      BLD   103;
      A     Q    216.4;
      =     L      1.1;
      BLD   103;
      A     Q    216.5;
      =     L      1.2;
      BLD   103;
      AN    M    504.0;
      AN    M    504.1;
      AN    M   6060.0;
      AN    M   6260.0;
      AN    M   6280.0;
      AN    M    504.2;
      A     M    500.2;
      =     L      1.3;
      BLD   103;
      A(    ;
      O     I      0.1;
      O     M   4120.1;
      )     ;
      =     L      1.5;
      BLD   103;
      A     M      0.5;
      =     L      1.6;
      BLD   103;
      CALL #S705_LM_DC_1ST_CLAMP2 (
           Enable_Aux               := L      0.0,
           Adv_Amount               := 2,
           Ret_Amount               := 2,
           LS_Adv1                  := L      0.1,
           LS_Ret1                  := L      0.2,
           LS_Adv2                  := L      0.3,
           LS_Ret2                  := L      0.4,
           SOL_Adv                  := L      1.1,
           SOL_Ret                  := L      1.2,
           M_Ready                  := L      1.3,
           T_CHK1                   := T#4S,
           T_CHK2                   := T#4S,
           PB_Error_Rst             := L      1.5,
           M_FLICK                  := L      1.6,
           M_Adv_Err                := M    650.4,
           M_Ret_Err                := M    650.5,
           Visu_Adv                 := DB51.DBW   48,
           Visu_Ret                 := DB51.DBW   50);
      NOP   0;
NETWORK
TITLE =
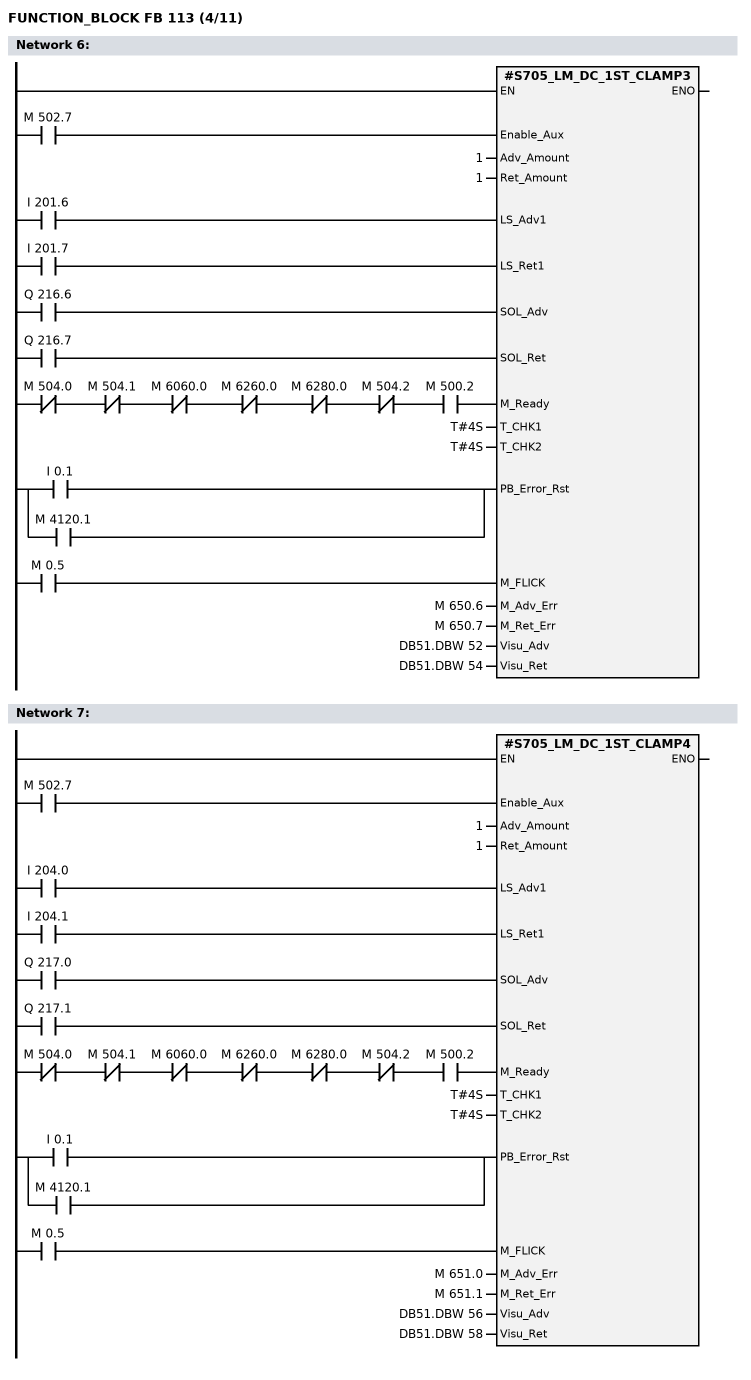

      A     M    502.7;
      =     L      0.0;
      BLD   103;
      A     I    201.6;
      =     L      0.1;
      BLD   103;
      A     I    201.7;
      =     L      0.2;
      BLD   103;
      A     Q    216.6;
      =     L      1.1;
      BLD   103;
      A     Q    216.7;
      =     L      1.2;
      BLD   103;
      AN    M    504.0;
      AN    M    504.1;
      AN    M   6060.0;
      AN    M   6260.0;
      AN    M   6280.0;
      AN    M    504.2;
      A     M    500.2;
      =     L      1.3;
      BLD   103;
      A(    ;
      O     I      0.1;
      O     M   4120.1;
      )     ;
      =     L      1.5;
      BLD   103;
      A     M      0.5;
      =     L      1.6;
      BLD   103;
      CALL #S705_LM_DC_1ST_CLAMP3 (
           Enable_Aux               := L      0.0,
           Adv_Amount               := 1,
           Ret_Amount               := 1,
           LS_Adv1                  := L      0.1,
           LS_Ret1                  := L      0.2,
           SOL_Adv                  := L      1.1,
           SOL_Ret                  := L      1.2,
           M_Ready                  := L      1.3,
           T_CHK1                   := T#4S,
           T_CHK2                   := T#4S,
           PB_Error_Rst             := L      1.5,
           M_FLICK                  := L      1.6,
           M_Adv_Err                := M    650.6,
           M_Ret_Err                := M    650.7,
           Visu_Adv                 := DB51.DBW   52,
           Visu_Ret                 := DB51.DBW   54);
      NOP   0;
NETWORK
TITLE =

      A     M    502.7;
      =     L      0.0;
      BLD   103;
      A     I    204.0;
      =     L      0.1;
      BLD   103;
      A     I    204.1;
      =     L      0.2;
      BLD   103;
      A     Q    217.0;
      =     L      1.1;
      BLD   103;
      A     Q    217.1;
      =     L      1.2;
      BLD   103;
      AN    M    504.0;
      AN    M    504.1;
      AN    M   6060.0;
      AN    M   6260.0;
      AN    M   6280.0;
      AN    M    504.2;
      A     M    500.2;
      =     L      1.3;
      BLD   103;
      A(    ;
      O     I      0.1;
      O     M   4120.1;
      )     ;
      =     L      1.5;
      BLD   103;
      A     M      0.5;
      =     L      1.6;
      BLD   103;
      CALL #S705_LM_DC_1ST_CLAMP4 (
           Enable_Aux               := L      0.0,
           Adv_Amount               := 1,
           Ret_Amount               := 1,
           LS_Adv1                  := L      0.1,
           LS_Ret1                  := L      0.2,
           SOL_Adv                  := L      1.1,
           SOL_Ret                  := L      1.2,
           M_Ready                  := L      1.3,
           T_CHK1                   := T#4S,
           T_CHK2                   := T#4S,
           PB_Error_Rst             := L      1.5,
           M_FLICK                  := L      1.6,
           M_Adv_Err                := M    651.0,
           M_Ret_Err                := M    651.1,
           Visu_Adv                 := DB51.DBW   56,
           Visu_Ret                 := DB51.DBW   58);
      NOP   0;
NETWORK
TITLE =
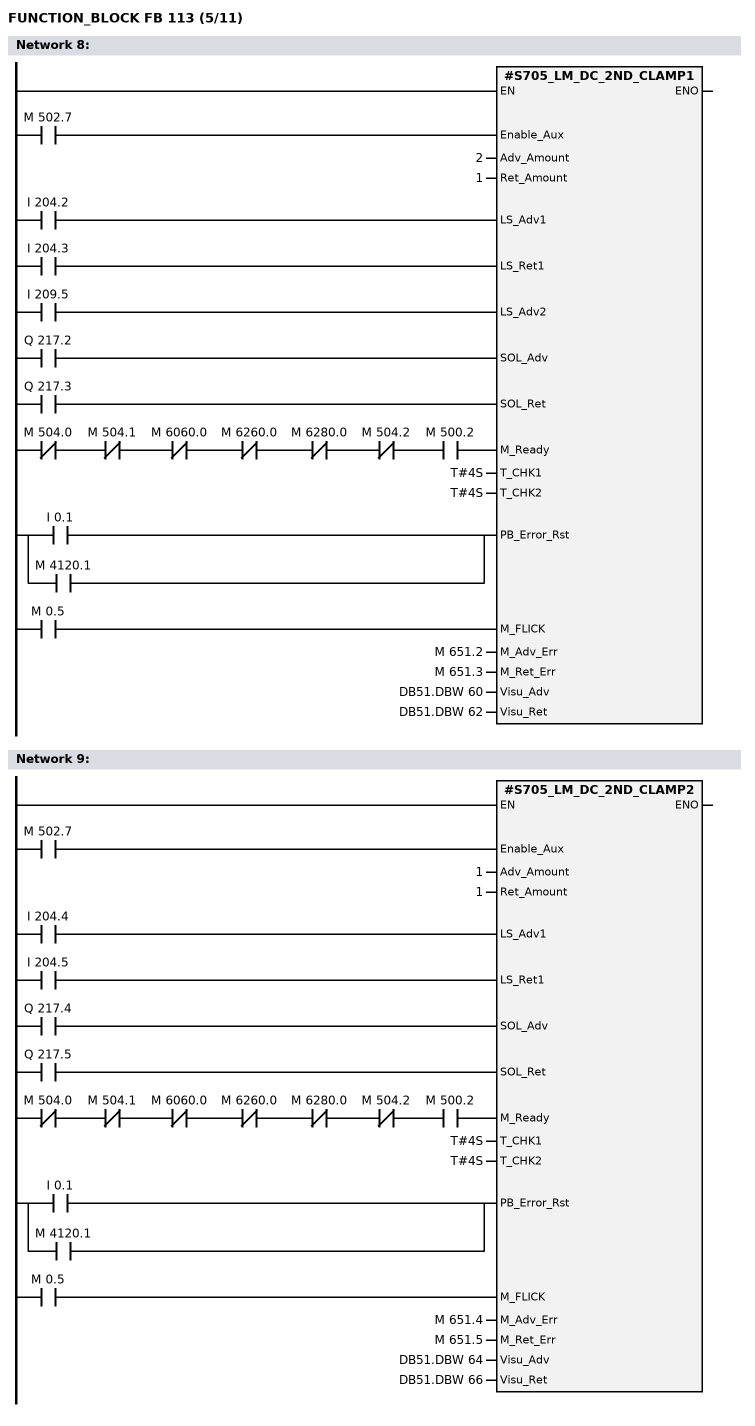

      A     M    502.7;
      =     L      0.0;
      BLD   103;
      A     I    204.2;
      =     L      0.1;
      BLD   103;
      A     I    204.3;
      =     L      0.2;
      BLD   103;
      A     I    209.5;
      =     L      0.3;
      BLD   103;
      A     Q    217.2;
      =     L      1.1;
      BLD   103;
      A     Q    217.3;
      =     L      1.2;
      BLD   103;
      AN    M    504.0;
      AN    M    504.1;
      AN    M   6060.0;
      AN    M   6260.0;
      AN    M   6280.0;
      AN    M    504.2;
      A     M    500.2;
      =     L      1.3;
      BLD   103;
      A(    ;
      O     I      0.1;
      O     M   4120.1;
      )     ;
      =     L      1.5;
      BLD   103;
      A     M      0.5;
      =     L      1.6;
      BLD   103;
      CALL #S705_LM_DC_2ND_CLAMP1 (
           Enable_Aux               := L      0.0,
           Adv_Amount               := 2,
           Ret_Amount               := 1,
           LS_Adv1                  := L      0.1,
           LS_Ret1                  := L      0.2,
           LS_Adv2                  := L      0.3,
           SOL_Adv                  := L      1.1,
           SOL_Ret                  := L      1.2,
           M_Ready                  := L      1.3,
           T_CHK1                   := T#4S,
           T_CHK2                   := T#4S,
           PB_Error_Rst             := L      1.5,
           M_FLICK                  := L      1.6,
           M_Adv_Err                := M    651.2,
           M_Ret_Err                := M    651.3,
           Visu_Adv                 := DB51.DBW   60,
           Visu_Ret                 := DB51.DBW   62);
      NOP   0;
NETWORK
TITLE =

      A     M    502.7;
      =     L      0.0;
      BLD   103;
      A     I    204.4;
      =     L      0.1;
      BLD   103;
      A     I    204.5;
      =     L      0.2;
      BLD   103;
      A     Q    217.4;
      =     L      1.1;
      BLD   103;
      A     Q    217.5;
      =     L      1.2;
      BLD   103;
      AN    M    504.0;
      AN    M    504.1;
      AN    M   6060.0;
      AN    M   6260.0;
      AN    M   6280.0;
      AN    M    504.2;
      A     M    500.2;
      =     L      1.3;
      BLD   103;
      A(    ;
      O     I      0.1;
      O     M   4120.1;
      )     ;
      =     L      1.5;
      BLD   103;
      A     M      0.5;
      =     L      1.6;
      BLD   103;
      CALL #S705_LM_DC_2ND_CLAMP2 (
           Enable_Aux               := L      0.0,
           Adv_Amount               := 1,
           Ret_Amount               := 1,
           LS_Adv1                  := L      0.1,
           LS_Ret1                  := L      0.2,
           SOL_Adv                  := L      1.1,
           SOL_Ret                  := L      1.2,
           M_Ready                  := L      1.3,
           T_CHK1                   := T#4S,
           T_CHK2                   := T#4S,
           PB_Error_Rst             := L      1.5,
           M_FLICK                  := L      1.6,
           M_Adv_Err                := M    651.4,
           M_Ret_Err                := M    651.5,
           Visu_Adv                 := DB51.DBW   64,
           Visu_Ret                 := DB51.DBW   66);
      NOP   0;
NETWORK
TITLE =
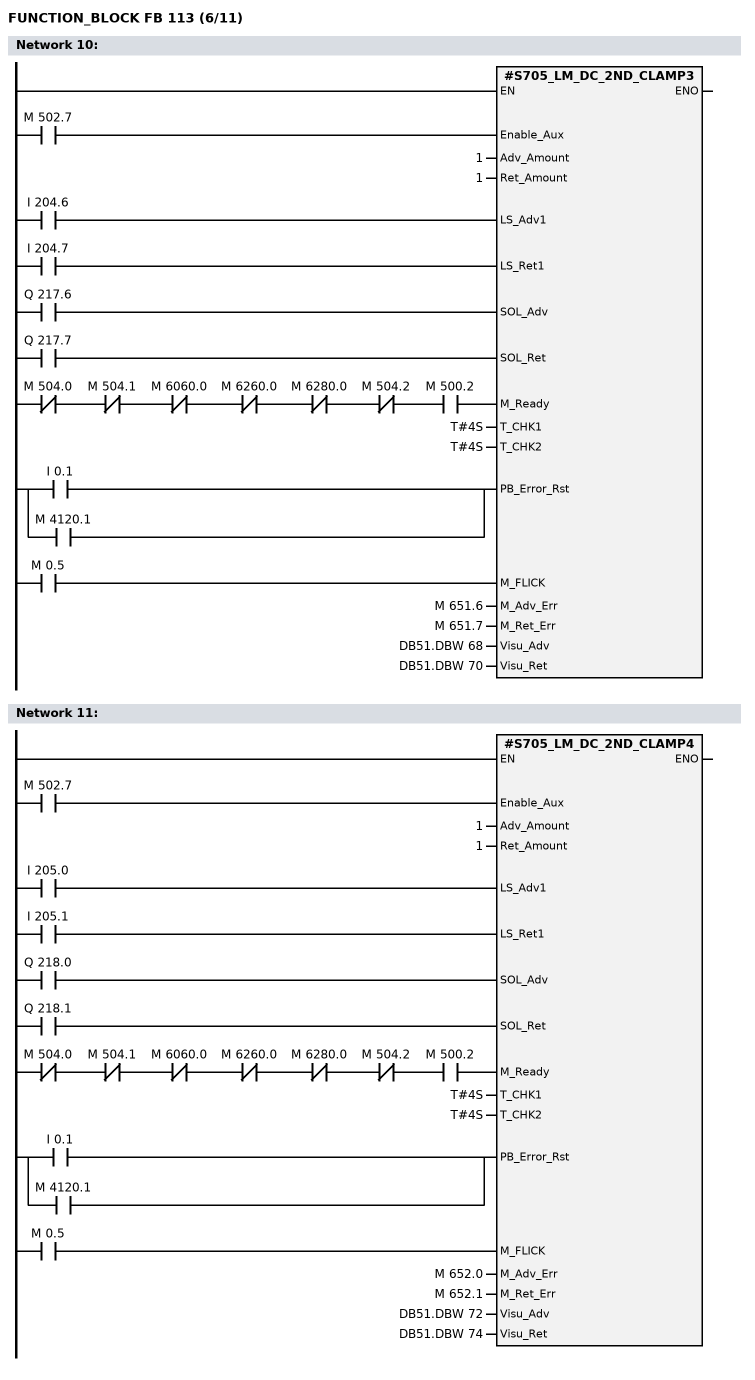

      A     M    502.7;
      =     L      0.0;
      BLD   103;
      A     I    204.6;
      =     L      0.1;
      BLD   103;
      A     I    204.7;
      =     L      0.2;
      BLD   103;
      A     Q    217.6;
      =     L      1.1;
      BLD   103;
      A     Q    217.7;
      =     L      1.2;
      BLD   103;
      AN    M    504.0;
      AN    M    504.1;
      AN    M   6060.0;
      AN    M   6260.0;
      AN    M   6280.0;
      AN    M    504.2;
      A     M    500.2;
      =     L      1.3;
      BLD   103;
      A(    ;
      O     I      0.1;
      O     M   4120.1;
      )     ;
      =     L      1.5;
      BLD   103;
      A     M      0.5;
      =     L      1.6;
      BLD   103;
      CALL #S705_LM_DC_2ND_CLAMP3 (
           Enable_Aux               := L      0.0,
           Adv_Amount               := 1,
           Ret_Amount               := 1,
           LS_Adv1                  := L      0.1,
           LS_Ret1                  := L      0.2,
           SOL_Adv                  := L      1.1,
           SOL_Ret                  := L      1.2,
           M_Ready                  := L      1.3,
           T_CHK1                   := T#4S,
           T_CHK2                   := T#4S,
           PB_Error_Rst             := L      1.5,
           M_FLICK                  := L      1.6,
           M_Adv_Err                := M    651.6,
           M_Ret_Err                := M    651.7,
           Visu_Adv                 := DB51.DBW   68,
           Visu_Ret                 := DB51.DBW   70);
      NOP   0;
NETWORK
TITLE =

      A     M    502.7;
      =     L      0.0;
      BLD   103;
      A     I    205.0;
      =     L      0.1;
      BLD   103;
      A     I    205.1;
      =     L      0.2;
      BLD   103;
      A     Q    218.0;
      =     L      1.1;
      BLD   103;
      A     Q    218.1;
      =     L      1.2;
      BLD   103;
      AN    M    504.0;
      AN    M    504.1;
      AN    M   6060.0;
      AN    M   6260.0;
      AN    M   6280.0;
      AN    M    504.2;
      A     M    500.2;
      =     L      1.3;
      BLD   103;
      A(    ;
      O     I      0.1;
      O     M   4120.1;
      )     ;
      =     L      1.5;
      BLD   103;
      A     M      0.5;
      =     L      1.6;
      BLD   103;
      CALL #S705_LM_DC_2ND_CLAMP4 (
           Enable_Aux               := L      0.0,
           Adv_Amount               := 1,
           Ret_Amount               := 1,
           LS_Adv1                  := L      0.1,
           LS_Ret1                  := L      0.2,
           SOL_Adv                  := L      1.1,
           SOL_Ret                  := L      1.2,
           M_Ready                  := L      1.3,
           T_CHK1                   := T#4S,
           T_CHK2                   := T#4S,
           PB_Error_Rst             := L      1.5,
           M_FLICK                  := L      1.6,
           M_Adv_Err                := M    652.0,
           M_Ret_Err                := M    652.1,
           Visu_Adv                 := DB51.DBW   72,
           Visu_Ret                 := DB51.DBW   74);
      NOP   0;
NETWORK
TITLE =
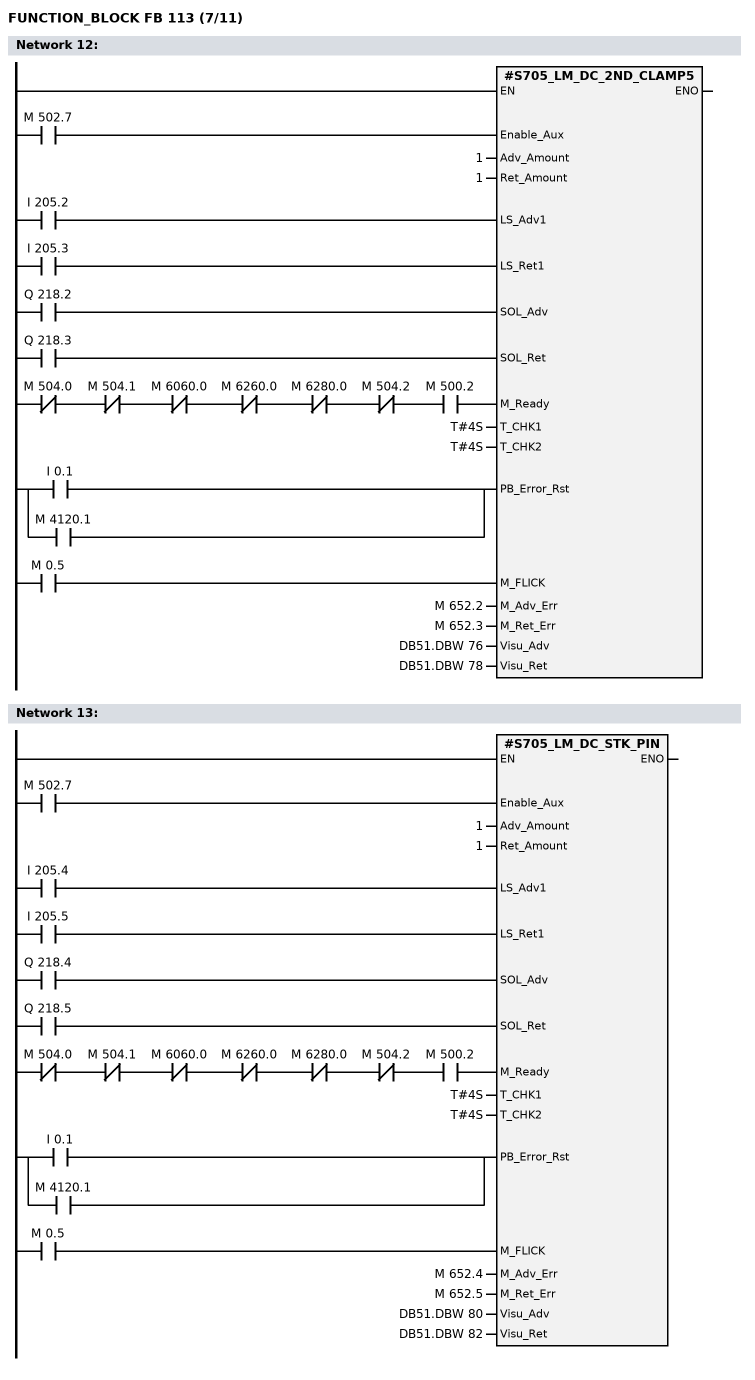

      A     M    502.7;
      =     L      0.0;
      BLD   103;
      A     I    205.2;
      =     L      0.1;
      BLD   103;
      A     I    205.3;
      =     L      0.2;
      BLD   103;
      A     Q    218.2;
      =     L      1.1;
      BLD   103;
      A     Q    218.3;
      =     L      1.2;
      BLD   103;
      AN    M    504.0;
      AN    M    504.1;
      AN    M   6060.0;
      AN    M   6260.0;
      AN    M   6280.0;
      AN    M    504.2;
      A     M    500.2;
      =     L      1.3;
      BLD   103;
      A(    ;
      O     I      0.1;
      O     M   4120.1;
      )     ;
      =     L      1.5;
      BLD   103;
      A     M      0.5;
      =     L      1.6;
      BLD   103;
      CALL #S705_LM_DC_2ND_CLAMP5 (
           Enable_Aux               := L      0.0,
           Adv_Amount               := 1,
           Ret_Amount               := 1,
           LS_Adv1                  := L      0.1,
           LS_Ret1                  := L      0.2,
           SOL_Adv                  := L      1.1,
           SOL_Ret                  := L      1.2,
           M_Ready                  := L      1.3,
           T_CHK1                   := T#4S,
           T_CHK2                   := T#4S,
           PB_Error_Rst             := L      1.5,
           M_FLICK                  := L      1.6,
           M_Adv_Err                := M    652.2,
           M_Ret_Err                := M    652.3,
           Visu_Adv                 := DB51.DBW   76,
           Visu_Ret                 := DB51.DBW   78);
      NOP   0;
NETWORK
TITLE =

      A     M    502.7;
      =     L      0.0;
      BLD   103;
      A     I    205.4;
      =     L      0.1;
      BLD   103;
      A     I    205.5;
      =     L      0.2;
      BLD   103;
      A     Q    218.4;
      =     L      1.1;
      BLD   103;
      A     Q    218.5;
      =     L      1.2;
      BLD   103;
      AN    M    504.0;
      AN    M    504.1;
      AN    M   6060.0;
      AN    M   6260.0;
      AN    M   6280.0;
      AN    M    504.2;
      A     M    500.2;
      =     L      1.3;
      BLD   103;
      A(    ;
      O     I      0.1;
      O     M   4120.1;
      )     ;
      =     L      1.5;
      BLD   103;
      A     M      0.5;
      =     L      1.6;
      BLD   103;
      CALL #S705_LM_DC_STK_PIN (
           Enable_Aux               := L      0.0,
           Adv_Amount               := 1,
           Ret_Amount               := 1,
           LS_Adv1                  := L      0.1,
           LS_Ret1                  := L      0.2,
           SOL_Adv                  := L      1.1,
           SOL_Ret                  := L      1.2,
           M_Ready                  := L      1.3,
           T_CHK1                   := T#4S,
           T_CHK2                   := T#4S,
           PB_Error_Rst             := L      1.5,
           M_FLICK                  := L      1.6,
           M_Adv_Err                := M    652.4,
           M_Ret_Err                := M    652.5,
           Visu_Adv                 := DB51.DBW   80,
           Visu_Ret                 := DB51.DBW   82);
      NOP   0;
NETWORK
TITLE =
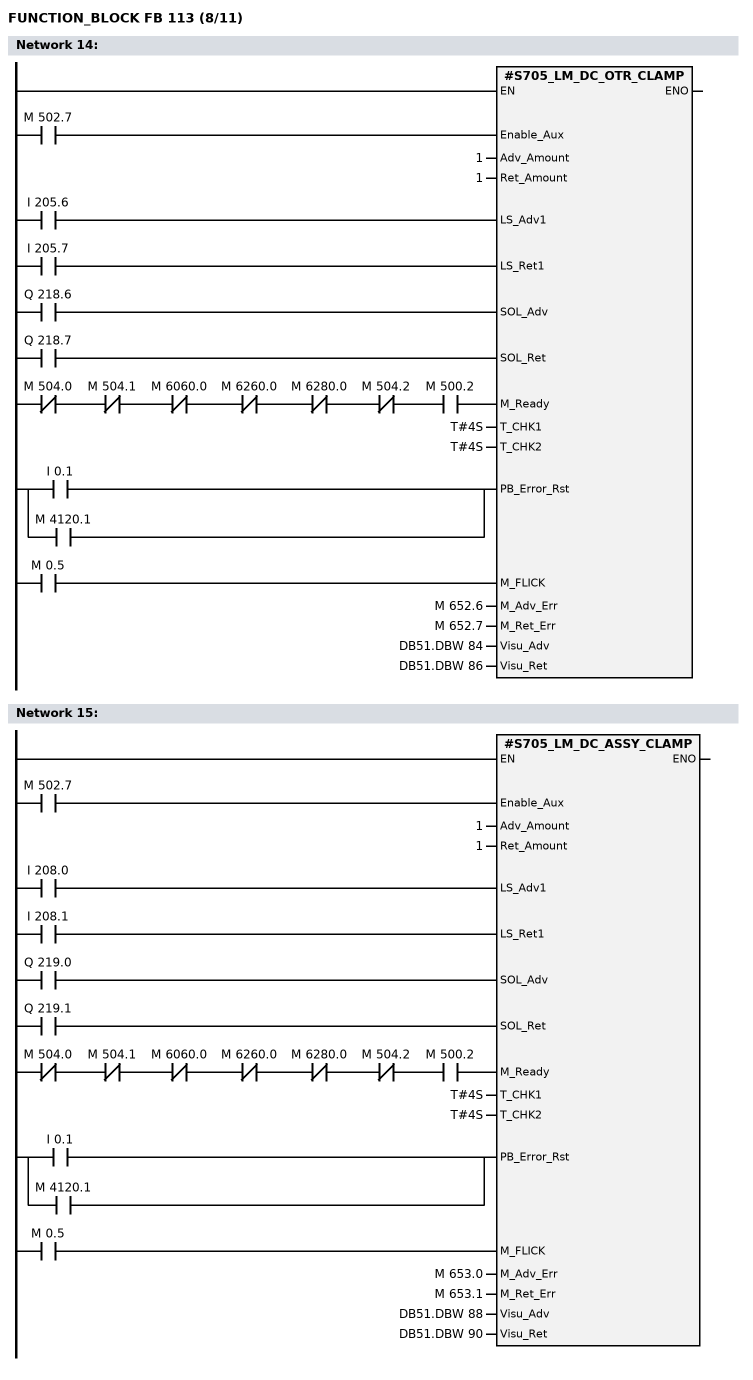

      A     M    502.7;
      =     L      0.0;
      BLD   103;
      A     I    205.6;
      =     L      0.1;
      BLD   103;
      A     I    205.7;
      =     L      0.2;
      BLD   103;
      A     Q    218.6;
      =     L      1.1;
      BLD   103;
      A     Q    218.7;
      =     L      1.2;
      BLD   103;
      AN    M    504.0;
      AN    M    504.1;
      AN    M   6060.0;
      AN    M   6260.0;
      AN    M   6280.0;
      AN    M    504.2;
      A     M    500.2;
      =     L      1.3;
      BLD   103;
      A(    ;
      O     I      0.1;
      O     M   4120.1;
      )     ;
      =     L      1.5;
      BLD   103;
      A     M      0.5;
      =     L      1.6;
      BLD   103;
      CALL #S705_LM_DC_OTR_CLAMP (
           Enable_Aux               := L      0.0,
           Adv_Amount               := 1,
           Ret_Amount               := 1,
           LS_Adv1                  := L      0.1,
           LS_Ret1                  := L      0.2,
           SOL_Adv                  := L      1.1,
           SOL_Ret                  := L      1.2,
           M_Ready                  := L      1.3,
           T_CHK1                   := T#4S,
           T_CHK2                   := T#4S,
           PB_Error_Rst             := L      1.5,
           M_FLICK                  := L      1.6,
           M_Adv_Err                := M    652.6,
           M_Ret_Err                := M    652.7,
           Visu_Adv                 := DB51.DBW   84,
           Visu_Ret                 := DB51.DBW   86);
      NOP   0;
NETWORK
TITLE =

      A     M    502.7;
      =     L      0.0;
      BLD   103;
      A     I    208.0;
      =     L      0.1;
      BLD   103;
      A     I    208.1;
      =     L      0.2;
      BLD   103;
      A     Q    219.0;
      =     L      1.1;
      BLD   103;
      A     Q    219.1;
      =     L      1.2;
      BLD   103;
      AN    M    504.0;
      AN    M    504.1;
      AN    M   6060.0;
      AN    M   6260.0;
      AN    M   6280.0;
      AN    M    504.2;
      A     M    500.2;
      =     L      1.3;
      BLD   103;
      A(    ;
      O     I      0.1;
      O     M   4120.1;
      )     ;
      =     L      1.5;
      BLD   103;
      A     M      0.5;
      =     L      1.6;
      BLD   103;
      CALL #S705_LM_DC_ASSY_CLAMP (
           Enable_Aux               := L      0.0,
           Adv_Amount               := 1,
           Ret_Amount               := 1,
           LS_Adv1                  := L      0.1,
           LS_Ret1                  := L      0.2,
           SOL_Adv                  := L      1.1,
           SOL_Ret                  := L      1.2,
           M_Ready                  := L      1.3,
           T_CHK1                   := T#4S,
           T_CHK2                   := T#4S,
           PB_Error_Rst             := L      1.5,
           M_FLICK                  := L      1.6,
           M_Adv_Err                := M    653.0,
           M_Ret_Err                := M    653.1,
           Visu_Adv                 := DB51.DBW   88,
           Visu_Ret                 := DB51.DBW   90);
      NOP   0;
NETWORK
TITLE =
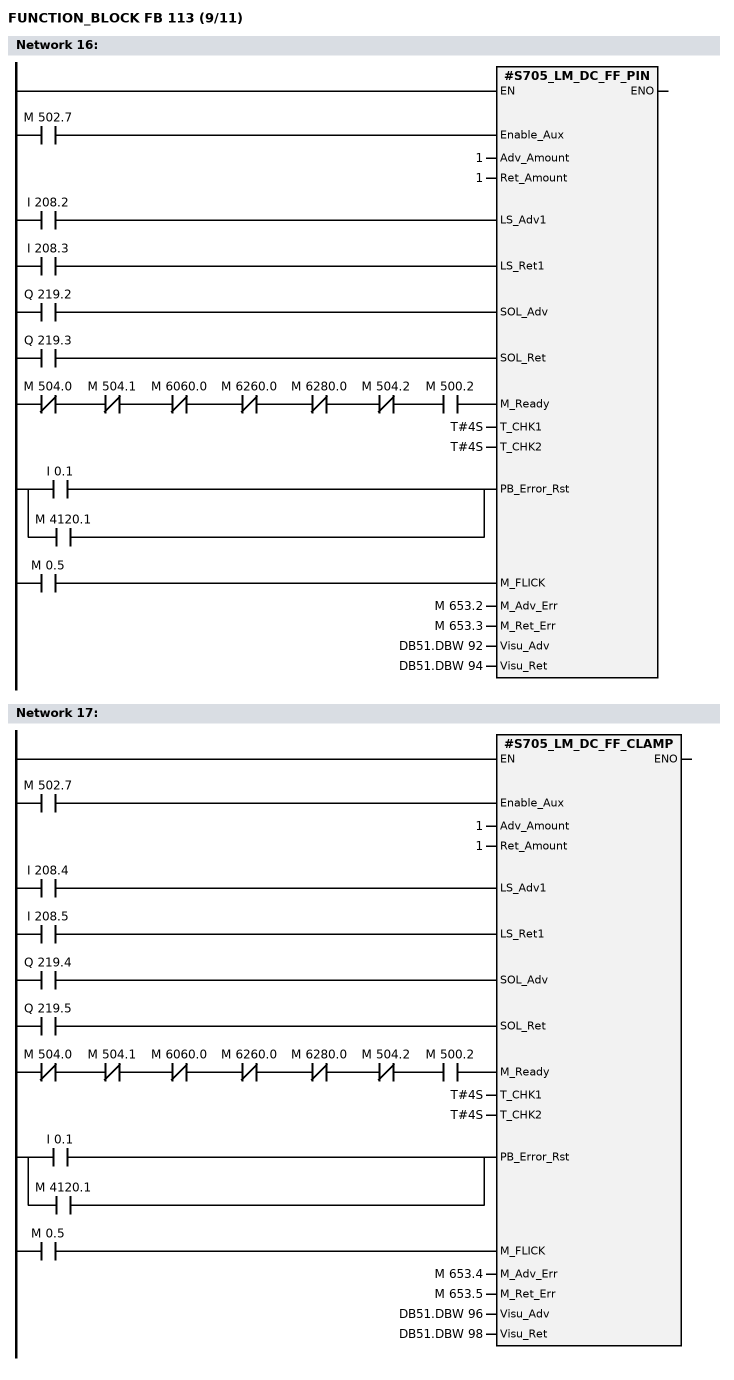

      A     M    502.7;
      =     L      0.0;
      BLD   103;
      A     I    208.2;
      =     L      0.1;
      BLD   103;
      A     I    208.3;
      =     L      0.2;
      BLD   103;
      A     Q    219.2;
      =     L      1.1;
      BLD   103;
      A     Q    219.3;
      =     L      1.2;
      BLD   103;
      AN    M    504.0;
      AN    M    504.1;
      AN    M   6060.0;
      AN    M   6260.0;
      AN    M   6280.0;
      AN    M    504.2;
      A     M    500.2;
      =     L      1.3;
      BLD   103;
      A(    ;
      O     I      0.1;
      O     M   4120.1;
      )     ;
      =     L      1.5;
      BLD   103;
      A     M      0.5;
      =     L      1.6;
      BLD   103;
      CALL #S705_LM_DC_FF_PIN (
           Enable_Aux               := L      0.0,
           Adv_Amount               := 1,
           Ret_Amount               := 1,
           LS_Adv1                  := L      0.1,
           LS_Ret1                  := L      0.2,
           SOL_Adv                  := L      1.1,
           SOL_Ret                  := L      1.2,
           M_Ready                  := L      1.3,
           T_CHK1                   := T#4S,
           T_CHK2                   := T#4S,
           PB_Error_Rst             := L      1.5,
           M_FLICK                  := L      1.6,
           M_Adv_Err                := M    653.2,
           M_Ret_Err                := M    653.3,
           Visu_Adv                 := DB51.DBW   92,
           Visu_Ret                 := DB51.DBW   94);
      NOP   0;
NETWORK
TITLE =

      A     M    502.7;
      =     L      0.0;
      BLD   103;
      A     I    208.4;
      =     L      0.1;
      BLD   103;
      A     I    208.5;
      =     L      0.2;
      BLD   103;
      A     Q    219.4;
      =     L      1.1;
      BLD   103;
      A     Q    219.5;
      =     L      1.2;
      BLD   103;
      AN    M    504.0;
      AN    M    504.1;
      AN    M   6060.0;
      AN    M   6260.0;
      AN    M   6280.0;
      AN    M    504.2;
      A     M    500.2;
      =     L      1.3;
      BLD   103;
      A(    ;
      O     I      0.1;
      O     M   4120.1;
      )     ;
      =     L      1.5;
      BLD   103;
      A     M      0.5;
      =     L      1.6;
      BLD   103;
      CALL #S705_LM_DC_FF_CLAMP (
           Enable_Aux               := L      0.0,
           Adv_Amount               := 1,
           Ret_Amount               := 1,
           LS_Adv1                  := L      0.1,
           LS_Ret1                  := L      0.2,
           SOL_Adv                  := L      1.1,
           SOL_Ret                  := L      1.2,
           M_Ready                  := L      1.3,
           T_CHK1                   := T#4S,
           T_CHK2                   := T#4S,
           PB_Error_Rst             := L      1.5,
           M_FLICK                  := L      1.6,
           M_Adv_Err                := M    653.4,
           M_Ret_Err                := M    653.5,
           Visu_Adv                 := DB51.DBW   96,
           Visu_Ret                 := DB51.DBW   98);
      NOP   0;
NETWORK
TITLE =
